REGION Network 13: Механізм крана
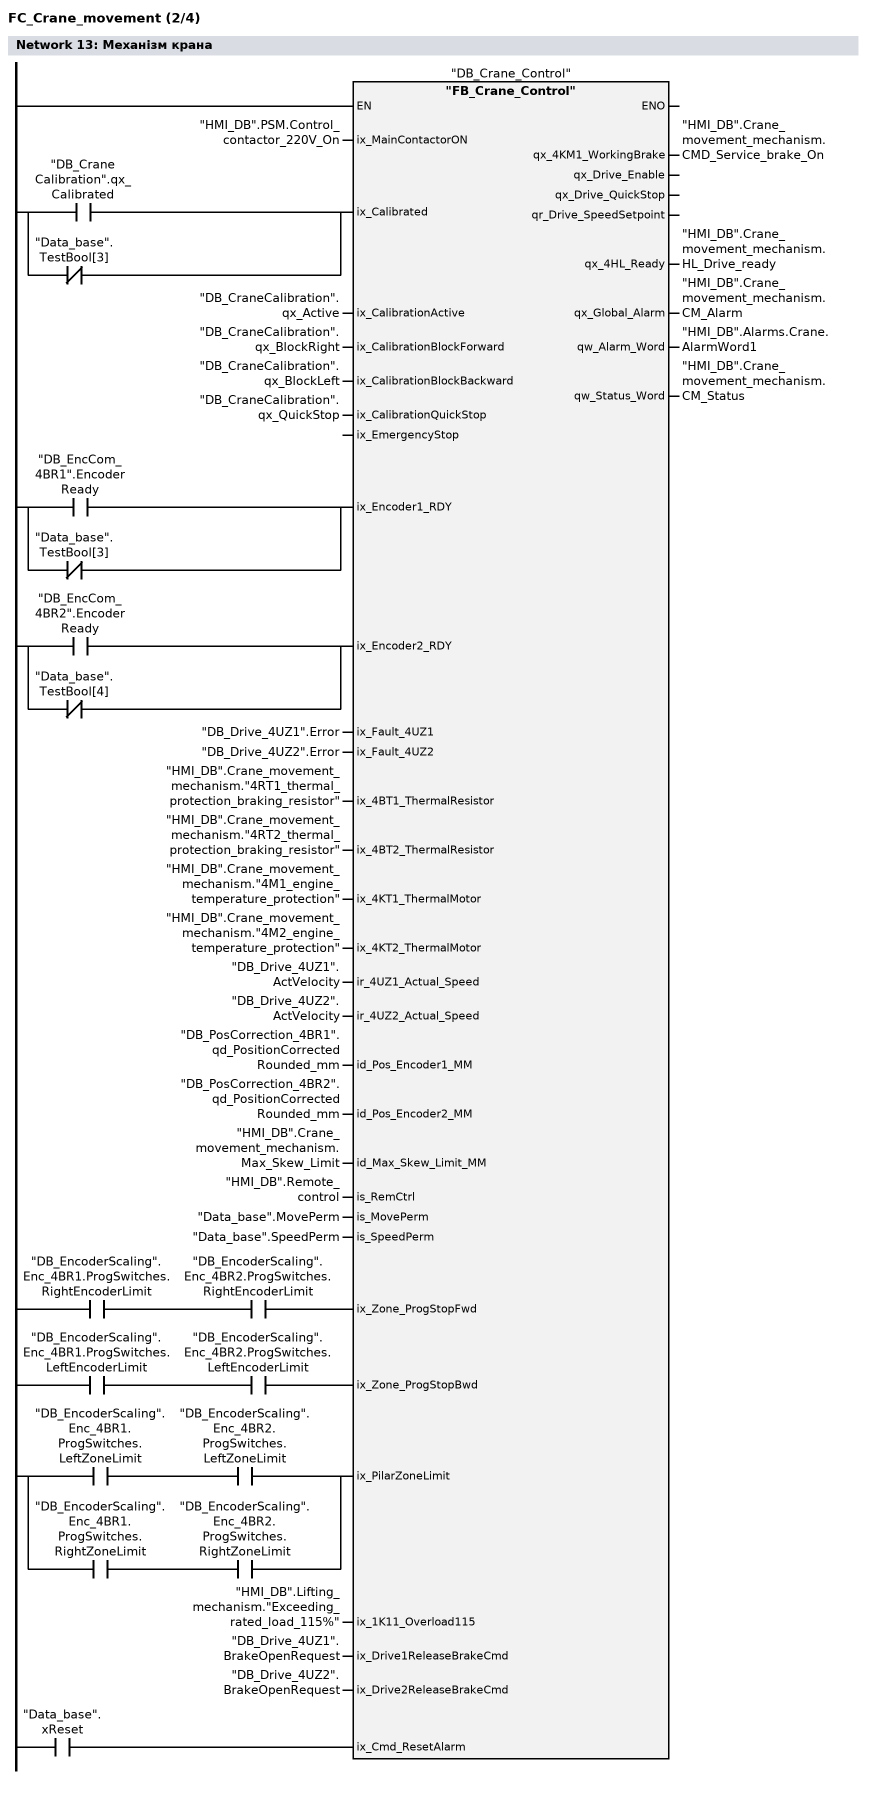
   RUNG wire#powerrail
      "DB_Crane_Control"(ix_Calibrated := wire#w1, ix_Encoder1_RDY := wire#w2, ix_Encoder2_RDY := wire#w3, ix_Zone_ProgStopFwd := wire#w4, ix_Zone_ProgStopBwd := wire#w5, ix_PilarZoneLimit := wire#w6, ix_Cmd_ResetAlarm := wire#w7, ix_MainContactorON := "HMI_DB".PSM.Control_contactor_220V_On, ix_CalibrationActive := "DB_CraneCalibration".qx_Active, ix_CalibrationBlockForward := "DB_CraneCalibration".qx_BlockRight, ix_CalibrationBlockBackward := "DB_CraneCalibration".qx_BlockLeft, ix_CalibrationQuickStop := "DB_CraneCalibration".qx_QuickStop, ix_EmergencyStop :=, ix_Fault_4UZ1 := "DB_Drive_4UZ1".Error, ix_Fault_4UZ2 := "DB_Drive_4UZ2".Error, ix_4BT1_ThermalResistor := "HMI_DB".Crane_movement_mechanism."4RT1_thermal_protection_braking_resistor", ix_4BT2_ThermalResistor := "HMI_DB".Crane_movement_mechanism."4RT2_thermal_protection_braking_resistor", ix_4KT1_ThermalMotor := "HMI_DB".Crane_movement_mechanism."4M1_engine_temperature_protection", ix_4KT2_ThermalMotor := "HMI_DB".Crane_movement_mechanism."4M2_engine_temperature_protection", ir_4UZ1_Actual_Speed := "DB_Drive_4UZ1".ActVelocity, ir_4UZ2_Actual_Speed := "DB_Drive_4UZ2".ActVelocity, id_Pos_Encoder1_MM := "DB_PosCorrection_4BR1".qd_PositionCorrectedRounded_mm, id_Pos_Encoder2_MM := "DB_PosCorrection_4BR2".qd_PositionCorrectedRounded_mm, id_Max_Skew_Limit_MM := "HMI_DB".Crane_movement_mechanism.Max_Skew_Limit, is_RemCtrl := "HMI_DB".Remote_control, is_MovePerm := "Data_base".MovePerm, is_SpeedPerm := "Data_base".SpeedPerm, ix_1K11_Overload115 := "HMI_DB".Lifting_mechanism."Exceeding_rated_load_115%", ix_Drive1ReleaseBrakeCmd := "DB_Drive_4UZ1".BrakeOpenRequest, ix_Drive2ReleaseBrakeCmd := "DB_Drive_4UZ2".BrakeOpenRequest, qx_4KM1_WorkingBrake => "HMI_DB".Crane_movement_mechanism.CMD_Service_brake_On, qx_Drive_Enable =>, qx_Drive_QuickStop =>, qr_Drive_SpeedSetpoint =>, qx_4HL_Ready => "HMI_DB".Crane_movement_mechanism.HL_Drive_ready, qx_Global_Alarm => "HMI_DB".Crane_movement_mechanism.CM_Alarm, qw_Alarm_Word => "HMI_DB".Alarms.Crane.AlarmWord1, qw_Status_Word => "HMI_DB".Crane_movement_mechanism.CM_Status)
   END_RUNG
   RUNG wire#powerrail
      Contact( "DB_CraneCalibration".qx_Calibrated )
   END_RUNG wire#w1
   RUNG wire#powerrail
      I_Contact( "Data_base".TestBool[3] )
   END_RUNG wire#w1
   RUNG wire#powerrail
      Contact( "DB_EncCom_4BR1".EncoderReady )
   END_RUNG wire#w2
   RUNG wire#powerrail
      I_Contact( "Data_base".TestBool[3] )
   END_RUNG wire#w2
   RUNG wire#powerrail
      Contact( "DB_EncCom_4BR2".EncoderReady )
   END_RUNG wire#w3
   RUNG wire#powerrail
      I_Contact( "Data_base".TestBool[4] )
   END_RUNG wire#w3
   RUNG wire#powerrail
      Contact( "DB_EncoderScaling".Enc_4BR1.ProgSwitches.RightEncoderLimit )
      Contact( "DB_EncoderScaling".Enc_4BR2.ProgSwitches.RightEncoderLimit )
   END_RUNG wire#w4
   RUNG wire#powerrail
      Contact( "DB_EncoderScaling".Enc_4BR1.ProgSwitches.LeftEncoderLimit )
      Contact( "DB_EncoderScaling".Enc_4BR2.ProgSwitches.LeftEncoderLimit )
   END_RUNG wire#w5
   RUNG wire#powerrail
      Contact( "DB_EncoderScaling".Enc_4BR1.ProgSwitches.LeftZoneLimit )
      Contact( "DB_EncoderScaling".Enc_4BR2.ProgSwitches.LeftZoneLimit )
   END_RUNG wire#w6
   RUNG wire#powerrail
      Contact( "DB_EncoderScaling".Enc_4BR1.ProgSwitches.RightZoneLimit )
      Contact( "DB_EncoderScaling".Enc_4BR2.ProgSwitches.RightZoneLimit )
   END_RUNG wire#w6
   RUNG wire#powerrail
      Contact( "Data_base".xReset )
   END_RUNG wire#w7
   // the same network as SCL:
   "DB_Crane_Control"(ix_MainContactorON := "HMI_DB".PSM.Control_contactor_220V_On,   // "FB_Crane_Control"
                      ix_Calibrated := "DB_CraneCalibration".qx_Calibrated OR NOT "Data_base".TestBool[3],
                      ix_CalibrationActive := "DB_CraneCalibration".qx_Active,
                      ix_CalibrationBlockForward := "DB_CraneCalibration".qx_BlockRight,
                      ix_CalibrationBlockBackward := "DB_CraneCalibration".qx_BlockLeft,
                      ix_CalibrationQuickStop := "DB_CraneCalibration".qx_QuickStop,
                      ix_Encoder1_RDY := "DB_EncCom_4BR1".EncoderReady OR NOT "Data_base".TestBool[3],
                      ix_Encoder2_RDY := "DB_EncCom_4BR2".EncoderReady OR NOT "Data_base".TestBool[4],
                      ix_Fault_4UZ1 := "DB_Drive_4UZ1".Error,
                      ix_Fault_4UZ2 := "DB_Drive_4UZ2".Error,
                      ix_4BT1_ThermalResistor := "HMI_DB".Crane_movement_mechanism."4RT1_thermal_protection_braking_resistor",
                      ix_4BT2_ThermalResistor := "HMI_DB".Crane_movement_mechanism."4RT2_thermal_protection_braking_resistor",
                      ix_4KT1_ThermalMotor := "HMI_DB".Crane_movement_mechanism."4M1_engine_temperature_protection",
                      ix_4KT2_ThermalMotor := "HMI_DB".Crane_movement_mechanism."4M2_engine_temperature_protection",
                      ir_4UZ1_Actual_Speed := "DB_Drive_4UZ1".ActVelocity,
                      ir_4UZ2_Actual_Speed := "DB_Drive_4UZ2".ActVelocity,
                      id_Pos_Encoder1_MM := "DB_PosCorrection_4BR1".qd_PositionCorrectedRounded_mm,
                      id_Pos_Encoder2_MM := "DB_PosCorrection_4BR2".qd_PositionCorrectedRounded_mm,
                      id_Max_Skew_Limit_MM := "HMI_DB".Crane_movement_mechanism.Max_Skew_Limit,
                      is_RemCtrl := "HMI_DB".Remote_control,
                      is_MovePerm := "Data_base".MovePerm,
                      is_SpeedPerm := "Data_base".SpeedPerm,
                      ix_Zone_ProgStopFwd := "DB_EncoderScaling".Enc_4BR1.ProgSwitches.RightEncoderLimit AND "DB_EncoderScaling".Enc_4BR2.ProgSwitches.RightEncoderLimit,
                      ix_Zone_ProgStopBwd := "DB_EncoderScaling".Enc_4BR1.ProgSwitches.LeftEncoderLimit AND "DB_EncoderScaling".Enc_4BR2.ProgSwitches.LeftEncoderLimit,
                      ix_PilarZoneLimit := ("DB_EncoderScaling".Enc_4BR1.ProgSwitches.LeftZoneLimit AND "DB_EncoderScaling".Enc_4BR2.ProgSwitches.LeftZoneLimit) OR ("DB_EncoderScaling".Enc_4BR1.ProgSwitches.RightZoneLimit AND "DB_EncoderScaling".Enc_4BR2.ProgSwitches.RightZoneLimit),
                      ix_1K11_Overload115 := "HMI_DB".Lifting_mechanism."Exceeding_rated_load_115%",
                      ix_Drive1ReleaseBrakeCmd := "DB_Drive_4UZ1".BrakeOpenRequest,
                      ix_Drive2ReleaseBrakeCmd := "DB_Drive_4UZ2".BrakeOpenRequest,
                      ix_Cmd_ResetAlarm := "Data_base".xReset,
                      qx_4KM1_WorkingBrake => "HMI_DB".Crane_movement_mechanism.CMD_Service_brake_On,
                      qx_4HL_Ready => "HMI_DB".Crane_movement_mechanism.HL_Drive_ready,
                      qx_Global_Alarm => "HMI_DB".Crane_movement_mechanism.CM_Alarm,
                      qw_Alarm_Word => "HMI_DB".Alarms.Crane.AlarmWord1,
                      qw_Status_Word => "HMI_DB".Crane_movement_mechanism.CM_Status);
END_REGION

REGION Network 14: Регістрація дій оператора
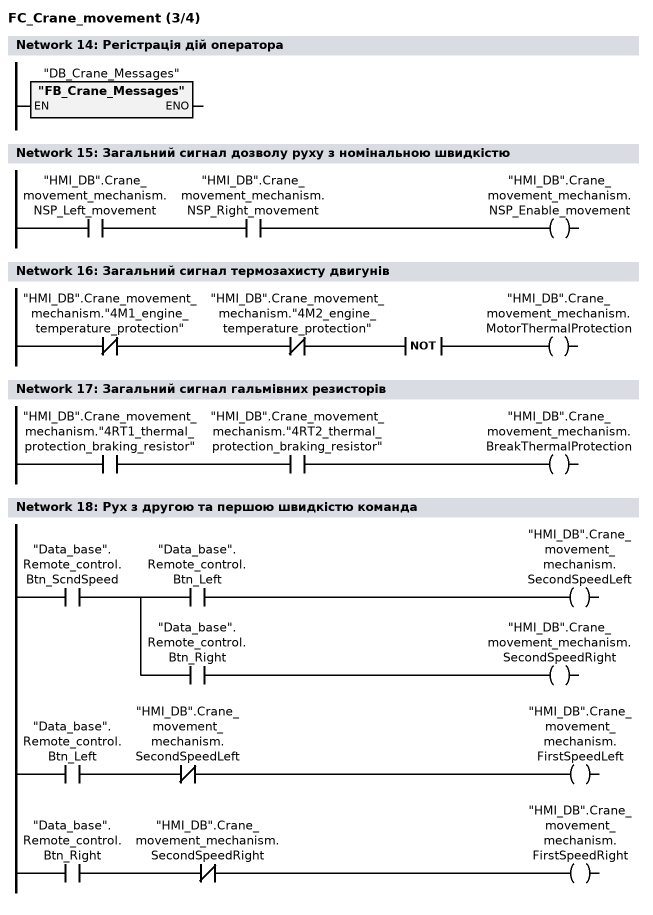
   RUNG wire#powerrail
      "DB_Crane_Messages"()
   END_RUNG
   // the same network as SCL:
   "DB_Crane_Messages"();   // "FB_Crane_Messages"
END_REGION

REGION Network 15: Загальний сигнал дозволу руху з номінальною швидкістю
   RUNG wire#powerrail
      Contact( "HMI_DB".Crane_movement_mechanism.NSP_Left_movement )
      Contact( "HMI_DB".Crane_movement_mechanism.NSP_Right_movement )
      Coil( "HMI_DB".Crane_movement_mechanism.NSP_Enable_movement )
   END_RUNG
   // the same network as SCL:
   "HMI_DB".Crane_movement_mechanism.NSP_Enable_movement := "HMI_DB".Crane_movement_mechanism.NSP_Left_movement AND "HMI_DB".Crane_movement_mechanism.NSP_Right_movement;
END_REGION

REGION Network 16: Загальний сигнал термозахисту двигунів
   RUNG wire#powerrail
      I_Contact( "HMI_DB".Crane_movement_mechanism."4M1_engine_temperature_protection" )
      I_Contact( "HMI_DB".Crane_movement_mechanism."4M2_engine_temperature_protection" )
      Not()
      Coil( "HMI_DB".Crane_movement_mechanism.MotorThermalProtection )
   END_RUNG
   // the same network as SCL:
   "HMI_DB".Crane_movement_mechanism.MotorThermalProtection := NOT (NOT "HMI_DB".Crane_movement_mechanism."4M1_engine_temperature_protection" AND NOT "HMI_DB".Crane_movement_mechanism."4M2_engine_temperature_protection");
END_REGION

REGION Network 17: Загальний сигнал гальмівних резисторів
   RUNG wire#powerrail
      Contact( "HMI_DB".Crane_movement_mechanism."4RT1_thermal_protection_braking_resistor" )
      Contact( "HMI_DB".Crane_movement_mechanism."4RT2_thermal_protection_braking_resistor" )
      Coil( "HMI_DB".Crane_movement_mechanism.BreakThermalProtection )
   END_RUNG
   // the same network as SCL:
   "HMI_DB".Crane_movement_mechanism.BreakThermalProtection := "HMI_DB".Crane_movement_mechanism."4RT1_thermal_protection_braking_resistor" AND "HMI_DB".Crane_movement_mechanism."4RT2_thermal_protection_braking_resistor";
END_REGION

REGION Network 18: Рух з другою та першою швидкістю команда
   RUNG wire#powerrail
      Contact( "Data_base".Remote_control.Btn_ScndSpeed )
      wire#w1
      Contact( "Data_base".Remote_control.Btn_Left )
      Coil( "HMI_DB".Crane_movement_mechanism.SecondSpeedLeft )
   END_RUNG
   RUNG wire#w1
      Contact( "Data_base".Remote_control.Btn_Right )
      Coil( "HMI_DB".Crane_movement_mechanism.SecondSpeedRight )
   END_RUNG
   RUNG wire#powerrail
      Contact( "Data_base".Remote_control.Btn_Left )
      I_Contact( "HMI_DB".Crane_movement_mechanism.SecondSpeedLeft )
      Coil( "HMI_DB".Crane_movement_mechanism.FirstSpeedLeft )
   END_RUNG
   RUNG wire#powerrail
      Contact( "Data_base".Remote_control.Btn_Right )
      I_Contact( "HMI_DB".Crane_movement_mechanism.SecondSpeedRight )
      Coil( "HMI_DB".Crane_movement_mechanism.FirstSpeedRight )
   END_RUNG
   // the same network as SCL:
   "HMI_DB".Crane_movement_mechanism.SecondSpeedLeft := "Data_base".Remote_control.Btn_ScndSpeed AND "Data_base".Remote_control.Btn_Left;
   "HMI_DB".Crane_movement_mechanism.SecondSpeedRight := "Data_base".Remote_control.Btn_ScndSpeed AND "Data_base".Remote_control.Btn_Right;
   "HMI_DB".Crane_movement_mechanism.FirstSpeedLeft := "Data_base".Remote_control.Btn_Left AND NOT "HMI_DB".Crane_movement_mechanism.SecondSpeedLeft;
   "HMI_DB".Crane_movement_mechanism.FirstSpeedRight := "Data_base".Remote_control.Btn_Right AND NOT "HMI_DB".Crane_movement_mechanism.SecondSpeedRight;
END_REGION

REGION Network 19: Формування попереджень калібровки
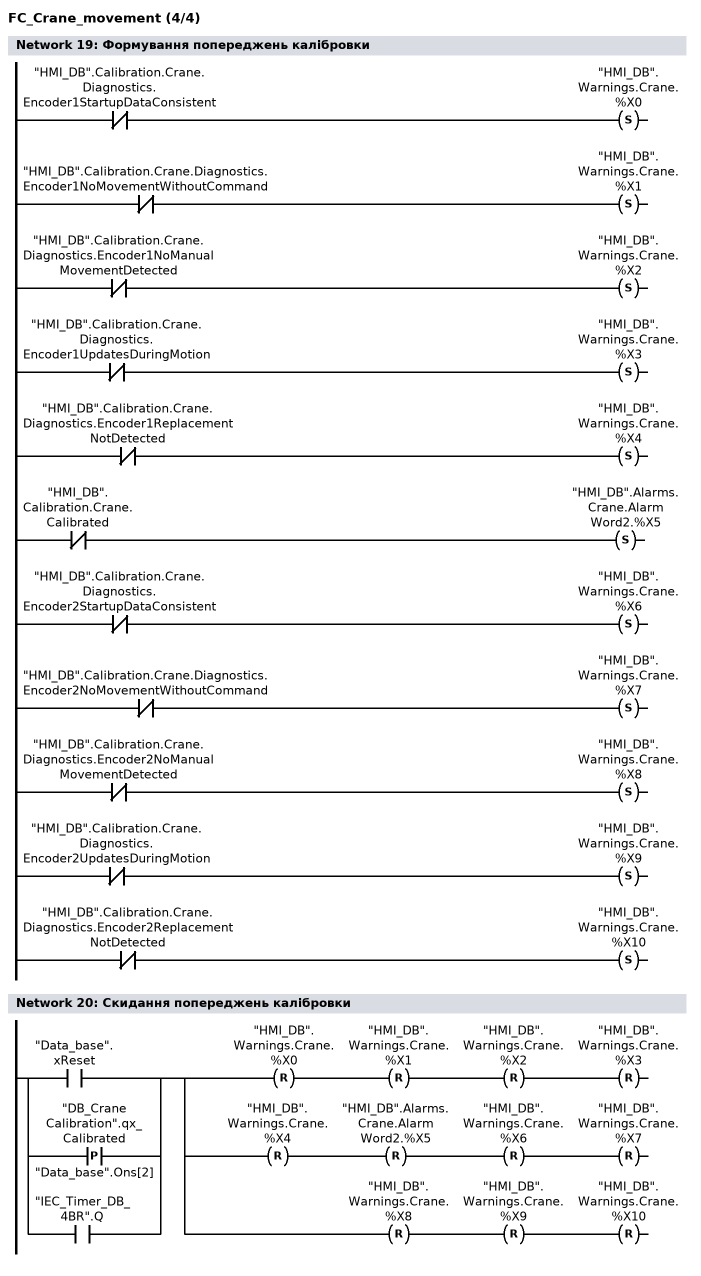
   RUNG wire#powerrail
      I_Contact( "HMI_DB".Calibration.Crane.Diagnostics.Encoder1StartupDataConsistent )
      S_Coil( "HMI_DB".Warnings.Crane.%X0 )
   END_RUNG
   RUNG wire#powerrail
      I_Contact( "HMI_DB".Calibration.Crane.Diagnostics.Encoder1NoMovementWithoutCommand )
      S_Coil( "HMI_DB".Warnings.Crane.%X1 )
   END_RUNG
   RUNG wire#powerrail
      I_Contact( "HMI_DB".Calibration.Crane.Diagnostics.Encoder1NoManualMovementDetected )
      S_Coil( "HMI_DB".Warnings.Crane.%X2 )
   END_RUNG
   RUNG wire#powerrail
      I_Contact( "HMI_DB".Calibration.Crane.Diagnostics.Encoder1UpdatesDuringMotion )
      S_Coil( "HMI_DB".Warnings.Crane.%X3 )
   END_RUNG
   RUNG wire#powerrail
      I_Contact( "HMI_DB".Calibration.Crane.Diagnostics.Encoder1ReplacementNotDetected )
      S_Coil( "HMI_DB".Warnings.Crane.%X4 )
   END_RUNG
   RUNG wire#powerrail
      I_Contact( "HMI_DB".Calibration.Crane.Calibrated )
      S_Coil( "HMI_DB".Alarms.Crane.AlarmWord2.%X5 )
   END_RUNG
   RUNG wire#powerrail
      I_Contact( "HMI_DB".Calibration.Crane.Diagnostics.Encoder2StartupDataConsistent )
      S_Coil( "HMI_DB".Warnings.Crane.%X6 )
   END_RUNG
   RUNG wire#powerrail
      I_Contact( "HMI_DB".Calibration.Crane.Diagnostics.Encoder2NoMovementWithoutCommand )
      S_Coil( "HMI_DB".Warnings.Crane.%X7 )
   END_RUNG
   RUNG wire#powerrail
      I_Contact( "HMI_DB".Calibration.Crane.Diagnostics.Encoder2NoManualMovementDetected )
      S_Coil( "HMI_DB".Warnings.Crane.%X8 )
   END_RUNG
   RUNG wire#powerrail
      I_Contact( "HMI_DB".Calibration.Crane.Diagnostics.Encoder2UpdatesDuringMotion )
      S_Coil( "HMI_DB".Warnings.Crane.%X9 )
   END_RUNG
   RUNG wire#powerrail
      I_Contact( "HMI_DB".Calibration.Crane.Diagnostics.Encoder2ReplacementNotDetected )
      S_Coil( "HMI_DB".Warnings.Crane.%X10 )
   END_RUNG
   // the same network as SCL:
   IF NOT "HMI_DB".Calibration.Crane.Diagnostics.Encoder1StartupDataConsistent THEN
       "HMI_DB".Warnings.Crane.%X0 := TRUE;
   END_IF;
   IF NOT "HMI_DB".Calibration.Crane.Diagnostics.Encoder1NoMovementWithoutCommand THEN
       "HMI_DB".Warnings.Crane.%X1 := TRUE;
   END_IF;
   IF NOT "HMI_DB".Calibration.Crane.Diagnostics.Encoder1NoManualMovementDetected THEN
       "HMI_DB".Warnings.Crane.%X2 := TRUE;
   END_IF;
   IF NOT "HMI_DB".Calibration.Crane.Diagnostics.Encoder1UpdatesDuringMotion THEN
       "HMI_DB".Warnings.Crane.%X3 := TRUE;
   END_IF;
   IF NOT "HMI_DB".Calibration.Crane.Diagnostics.Encoder1ReplacementNotDetected THEN
       "HMI_DB".Warnings.Crane.%X4 := TRUE;
   END_IF;
   IF NOT "HMI_DB".Calibration.Crane.Calibrated THEN "HMI_DB".Alarms.Crane.AlarmWord2.%X5 := TRUE; END_IF;
   IF NOT "HMI_DB".Calibration.Crane.Diagnostics.Encoder2StartupDataConsistent THEN
       "HMI_DB".Warnings.Crane.%X6 := TRUE;
   END_IF;
   IF NOT "HMI_DB".Calibration.Crane.Diagnostics.Encoder2NoMovementWithoutCommand THEN
       "HMI_DB".Warnings.Crane.%X7 := TRUE;
   END_IF;
   IF NOT "HMI_DB".Calibration.Crane.Diagnostics.Encoder2NoManualMovementDetected THEN
       "HMI_DB".Warnings.Crane.%X8 := TRUE;
   END_IF;
   IF NOT "HMI_DB".Calibration.Crane.Diagnostics.Encoder2UpdatesDuringMotion THEN
       "HMI_DB".Warnings.Crane.%X9 := TRUE;
   END_IF;
   IF NOT "HMI_DB".Calibration.Crane.Diagnostics.Encoder2ReplacementNotDetected THEN
       "HMI_DB".Warnings.Crane.%X10 := TRUE;
   END_IF;
END_REGION

REGION Network 20: Скидання попереджень калібровки
   RUNG wire#powerrail
      Contact( "Data_base".xReset )
      wire#w1
      R_Coil( "HMI_DB".Warnings.Crane.%X0 )
      R_Coil( "HMI_DB".Warnings.Crane.%X1 )
      R_Coil( "HMI_DB".Warnings.Crane.%X2 )
      R_Coil( "HMI_DB".Warnings.Crane.%X3 )
   END_RUNG
   RUNG wire#powerrail
      P_Contact(operand := "DB_CraneCalibration".qx_Calibrated, bit := "Data_base".Ons[2])
   END_RUNG wire#w1
   RUNG wire#powerrail
      Contact( "IEC_Timer_DB_4BR".Q )
   END_RUNG wire#w1
   RUNG wire#w1
      R_Coil( "HMI_DB".Warnings.Crane.%X4 )
      R_Coil( "HMI_DB".Alarms.Crane.AlarmWord2.%X5 )
      R_Coil( "HMI_DB".Warnings.Crane.%X6 )
      R_Coil( "HMI_DB".Warnings.Crane.%X7 )
   END_RUNG
   RUNG wire#w1
      R_Coil( "HMI_DB".Warnings.Crane.%X8 )
      R_Coil( "HMI_DB".Warnings.Crane.%X9 )
      R_Coil( "HMI_DB".Warnings.Crane.%X10 )
   END_RUNG
   // the same network as SCL:
   #_w1 := "DB_CraneCalibration".qx_Calibrated AND NOT "Data_base".Ons[2];   // rising edge of "DB_CraneCalibration".qx_Calibrated
   "Data_base".Ons[2] := "DB_CraneCalibration".qx_Calibrated;
   IF "Data_base".xReset OR #_w1 OR "IEC_Timer_DB_4BR".Q THEN
       "HMI_DB".Warnings.Crane.%X0 := FALSE;
       "HMI_DB".Warnings.Crane.%X1 := FALSE;
       "HMI_DB".Warnings.Crane.%X2 := FALSE;
       "HMI_DB".Warnings.Crane.%X3 := FALSE;
       "HMI_DB".Warnings.Crane.%X4 := FALSE;
       "HMI_DB".Alarms.Crane.AlarmWord2.%X5 := FALSE;
       "HMI_DB".Warnings.Crane.%X6 := FALSE;
       "HMI_DB".Warnings.Crane.%X7 := FALSE;
       "HMI_DB".Warnings.Crane.%X8 := FALSE;
       "HMI_DB".Warnings.Crane.%X9 := FALSE;
       "HMI_DB".Warnings.Crane.%X10 := FALSE;
   END_IF;
END_REGION
END_FUNCTION

// folder: 50_Drives

FUNCTION_BLOCK "FB_S120_Tel220"   // FB51, SCL
{ S7_Optimized_Access := 'TRUE' }
VERSION : 0.1
   VAR_INPUT
      EnableAxis : Bool := FALSE;   // Дозвіл роботи осі / ПЧ
      AckError : Bool := FALSE;   // Квітування аварії ПЧ, обробляється по фронту
      SimMode : Bool := FALSE;   // TRUE = режим симуляції, обмін з реальним ПЧ не виконується
      HWID_Tel220 : Hw_Io := 0;   // Hardware ID Telegram 220 для читання та запису PZD
      SpeedSp : Real := 0.0;   // Завдання швидкості, об/хв
      TorqueLimit : Real := 100.0;   // Обмеження моменту, %
      QuickStop : Bool := FALSE;   // Команда Quick Stop / OFF3
      CoastStop : Bool := FALSE;   // Команда Coast Stop / OFF2
      BrakesReleased : Bool := FALSE;   // Зворотний зв'язок: робоче та вбудоване гальма розгальмовані
      SimTelIn : "UDT_S120_Tel220_In";   // Симульована telegram від ПЧ
   END_VAR
   VAR_OUTPUT
      AxisEnabled : Bool := FALSE;   // ПЧ увімкнений та робота дозволена
      Lockout : Bool := FALSE;   // ПЧ не готовий до роботи або є заборона вмикання
      ActVelocity : Real := 0.0;   // Фактична швидкість, об/хв
      SpeedSetpointFb : Real := 0.0;   // Зворотний зв'язок по завданню швидкості, об/хв
      ActCurrent : Real := 0.0;   // Фактичний струм, А
      ActTorque : Real := 0.0;   // Фактичний момент, Н·м
      ActPower : Real := 0.0;   // Поточна активна потужність, кВт
      LoadPower : Real := 0.0;   // Завантаження механізму по потужності, %
      BrakeOpenRequest : Bool := FALSE;   // ПЧ запитує відкриття гальма
      Error : Bool := FALSE;   // Помилка драйвера або аварія ПЧ
      Status : Word := W#16#0000;   // Статус драйвера, бітове слово
      DiagId : Word := W#16#0000;   // Код діагностики драйвера / обміну
      FaultCode : Word := W#16#0000;   // Код аварії ПЧ
      WarningCode : Word := W#16#0000;   // Код попередження ПЧ
      TelOut : "UDT_S120_Tel220_Out";   // Сформована telegram PLC -> ПЧ, також для симулятора
   END_VAR
   VAR
      TelIn : "UDT_S120_Tel220_In";   // Остання прийнята telegram ПЧ -> PLC
      BrakeStatus : "UDT_S120_BrakeStatus";   // Розшифрований статус гальма з r1229
      ReadOk : Bool := FALSE;   // Читання telegram виконано без помилки
      WriteOk : Bool := FALSE;   // Запис telegram виконано без помилки
      ReadStatus : Int := 0;   // Код повернення DPRD_DAT
      WriteStatus : Int := 0;   // Код повернення DPWR_DAT
      ReadyToSwitchOn : Bool := FALSE;   // ПЧ готовий до вмикання
      ReadyToOperate : Bool := FALSE;   // ПЧ готовий до роботи
      OperationEnabled : Bool := FALSE;   // Робота ПЧ дозволена
      DriveFault : Bool := FALSE;   // Є аварія ПЧ
      DriveWarning : Bool := FALSE;   // Є попередження ПЧ
      NoCoastStopActive : Bool := FALSE;   // OFF2 не активний
      NoQuickStopActive : Bool := FALSE;   // OFF3 / Quick Stop не активний
      SwitchingOnInhibit : Bool := FALSE;   // Активна заборона вмикання
      ControlRequested : Bool := FALSE;   // ПЧ запитує керування від PLC
      RefSpeed_Rpm : Real := 1000.0;   // Опорна швидкість p2000, об/хв
      RefCurrent_A : Real := 1.0;   // Опорний струм p2002, А
      RefTorque_Nm : Real := 100.0;   // Опорний момент p2003, Н·м
      RefPower_kW : Real := 1.0;   // Опорна потужність p2004, кВт
      MotorRatedPower_kW : Real := 1.0;   // Номінальна потужність двигуна, кВт
      ResetFaultOld : Bool := FALSE;   // Попередній стан команди квітування аварії
      AckPulseCounter : Int := 0;   // Лічильник тривалості імпульсу квітування
      AckPulseCycles : Int := 10;   // Тривалість імпульсу квітування в циклах OB
   END_VAR
   VAR_TEMP
      ResetFaultPulse : Bool;   // Імпульс квітування аварії
      SpeedRawReal : Real;   // Завдання швидкості у сирому форматі telegram
      TorqueLimitRawReal : Real;   // Обмеження моменту у сирому форматі telegram
      TorqueLimitUsedPct : Real;   // Використане значення обмеження моменту
      AbsPower_kW : Real;   // Модуль активної потужності
   END_VAR
BEGIN
   // ============================================================
   // 1. Формування імпульсу квітування аварії
   // ============================================================

   IF #AckError AND NOT #ResetFaultOld THEN
       #AckPulseCounter := #AckPulseCycles;
   END_IF;

   #ResetFaultOld := #AckError;

   IF #AckPulseCounter > 0 THEN
       #ResetFaultPulse := TRUE;
       #AckPulseCounter := #AckPulseCounter - 1;
   ELSE
       #ResetFaultPulse := FALSE;
   END_IF;

   // ============================================================
   // 2. Формування вихідної telegram PLC -> ПЧ
   // ============================================================

   #TelOut.STW1_BM := W#16#0000;
   #TelOut.NSOLL_B := 0;
   #TelOut.STW2_BM := W#16#0000;
   #TelOut.M_ADD := 0;
   #TelOut.M_LIM := 0;
   #TelOut.USER_1 := W#16#0000;
   #TelOut.USER_2 := W#16#0000;
   #TelOut.USER_3 := W#16#0000;
   #TelOut.USER_4 := W#16#0000;

   // ============================================================
   // Feedback стану гальм для SINAMICS
   // Використовується механізмом підйому 1UZ1
   // ============================================================

   // PZD7, USER_1 bit 0:
   // робоче гальмо 1MB1 розгальмоване
   #TelOut.STW2_BM.%X12 := #BrakesReleased;
   #TelOut.STW2_BM.%X13 := NOT #BrakesReleased;
   // ============================================================

   // STW1_BM, базове керування PROFIdrive
   // Біт 01 = OFF2 не активний
   #TelOut.STW1_BM.%X1 := NOT #CoastStop;

   // Біт 02 = OFF3 / Quick Stop не активний
   #TelOut.STW1_BM.%X2 := NOT #QuickStop;

   // Біт 10 = керування від PLC
   #TelOut.STW1_BM.%X10 := TRUE;


       // Біт 09 = Enable Speed Controller
       #TelOut.STW2_BM.%X9 := TRUE;

   //IF #EnableAxis AND NOT #QuickStop AND NOT #CoastStop THEN
       // Біт 00 = ON / OFF1
       #TelOut.STW1_BM.%X0 :=#EnableAxis;

       // Біт 03 = дозвіл роботи
       #TelOut.STW1_BM.%X3 := TRUE;

       // Біт 04 = дозвіл генератора рампи
       #TelOut.STW1_BM.%X4 := TRUE;

       // Біт 05 = продовження роботи генератора рампи
       #TelOut.STW1_BM.%X5 := TRUE;


       // Біт 06 = дозвіл завдання швидкості
       #TelOut.STW1_BM.%X6 := TRUE;
   //END_IF;

   // Біт 07 = квітування аварії ПЧ, імпульсом
   #TelOut.STW1_BM.%X7 := #ResetFaultPulse;


   // ============================================================
   // 3. Масштабування завдання швидкості
   // NSOLL_B є 32-бітовим нормалізованим значенням.
   // 16#40000000 = 1073741824 = 100 % RefSpeed_Rpm
   // ============================================================

   IF #EnableAxis
       AND NOT #QuickStop
       AND NOT #CoastStop
       AND (#RefSpeed_Rpm > 0.0)
   THEN
       #SpeedRawReal := (#SpeedSp / #RefSpeed_Rpm) * 1073741824.0;

       IF #SpeedRawReal > 2147483647.0 THEN
           #SpeedRawReal := 2147483647.0;
       ELSIF #SpeedRawReal < -2147483648.0 THEN
           #SpeedRawReal := -2147483648.0;
       END_IF;

       #TelOut.NSOLL_B := REAL_TO_DINT(#SpeedRawReal);
   ELSE
       #TelOut.NSOLL_B := 0;
   END_IF;

   // ============================================================
   // 4. Обмеження моменту
   // ============================================================

   IF #TorqueLimit > 0.0 THEN
       #TorqueLimitUsedPct := #TorqueLimit;
   ELSE
       #TorqueLimitUsedPct := 100.0;
   END_IF;

   #TorqueLimitRawReal := (#TorqueLimitUsedPct / 100.0) * 16384.0;

   IF #TorqueLimitRawReal > 32767.0 THEN
       #TorqueLimitRawReal := 32767.0;
   ELSIF #TorqueLimitRawReal < 0.0 THEN
       #TorqueLimitRawReal := 0.0;
   END_IF;

   #TelOut.M_LIM := REAL_TO_INT(#TorqueLimitRawReal);


   // ============================================================
   // 5. Запис telegram PLC -> ПЧ
   // Один HWID_Tel220 використовується для запису та читання
   // ============================================================

   //IF #SimMode THEN
   //    #WriteStatus := 0;
   //    #WriteOk := TRUE;
   //ELSE
    //   #WriteStatus := DPWR_DAT(
    //                            LADDR := #HWID_Tel220,
   //                             RECORD := #TelOut
    //   );
    //   #WriteOk := (#WriteStatus = 0);
   //END_IF;

   #WriteStatus := DPWR_DAT(
                            LADDR := #HWID_Tel220,
                            RECORD := #TelOut
   );
   #WriteOk := (#WriteStatus = 0);

   // ============================================================
   // 6. Читання telegram ПЧ -> PLC або симуляція
   // Один HWID_Tel220 використовується для запису та читання
   // ============================================================

   //IF #SimMode THEN
    //   #TelIn := #SimTelIn;
    //   #ReadStatus := 0;
   //    #ReadOk := TRUE;
   //ELSE
    //   #ReadStatus := DPRD_DAT(
    //                           LADDR := #HWID_Tel220,
    //                           RECORD => #TelIn
    //   );

    //   #ReadOk := (#ReadStatus = 0);
   //END_IF;
   #ReadStatus := DPRD_DAT(
                           LADDR := #HWID_Tel220,
                           RECORD => #TelIn
   );

   #ReadOk := (#ReadStatus = 0);

   // ============================================================
   // 7. Декодування ZSW1_BM
   // ============================================================

   #ReadyToSwitchOn := #TelIn.ZSW1_BM.%X0;
   #ReadyToOperate := #TelIn.ZSW1_BM.%X1;
   #OperationEnabled := #TelIn.ZSW1_BM.%X2;
   #DriveFault := #TelIn.ZSW1_BM.%X3;
   #NoCoastStopActive := #TelIn.ZSW1_BM.%X4;
   #NoQuickStopActive := #TelIn.ZSW1_BM.%X5;
   #SwitchingOnInhibit := #TelIn.ZSW1_BM.%X6;
   #DriveWarning := #TelIn.ZSW1_BM.%X7;
   #ControlRequested := #TelIn.ZSW1_BM.%X9;


   // ============================================================
   // 8. Основні статуси для зовнішньої логіки
   // ============================================================

   #AxisEnabled := #ReadOk
   AND #WriteOk
   AND #OperationEnabled
   AND NOT #DriveFault;

   #Lockout := (NOT #ReadOk)
   OR (NOT #WriteOk)
   OR #DriveFault
   OR #SwitchingOnInhibit
   OR (NOT #NoCoastStopActive)
   OR (NOT #NoQuickStopActive);

   #Error := (NOT #ReadOk)
   OR (NOT #WriteOk)
   OR #DriveFault;


   // ============================================================
   // 9. Коди fault / warning
   // ============================================================

   #FaultCode := #TelIn.FAULT_CODE;
   #WarningCode := #TelIn.WARN_CODE;


   // ============================================================
   // 10. Масштабування фактичних значень
   // ============================================================

   #ActVelocity := 0.0;
   #SpeedSetpointFb := 0.0;
   #ActCurrent := 0.0;
   #ActTorque := 0.0;
   #ActPower := 0.0;
   #LoadPower := 0.0;
   #AbsPower_kW := 0.0;

   IF #RefSpeed_Rpm > 0.0 THEN
       #ActVelocity := (INT_TO_REAL(#TelIn.NIST_A) / 16384.0) * #RefSpeed_Rpm;
       #SpeedSetpointFb := (INT_TO_REAL(#TelIn.NSET_FB) / 16384.0) * #RefSpeed_Rpm;
   END_IF;

   IF #RefCurrent_A > 0.0 THEN
       #ActCurrent := (INT_TO_REAL(#TelIn.IAIST) / 16384.0) * #RefCurrent_A;
   END_IF;

   IF #RefTorque_Nm > 0.0 THEN
       #ActTorque := (INT_TO_REAL(#TelIn.MIST) / 16384.0) * #RefTorque_Nm;
   END_IF;

   IF #RefPower_kW > 0.0 THEN
       #ActPower := (INT_TO_REAL(#TelIn.P_ACT) / 16384.0) * #RefPower_kW;
   END_IF;

   IF #ActPower < 0.0 THEN
       #AbsPower_kW := - #ActPower;
   ELSE
       #AbsPower_kW := #ActPower;
   END_IF;

   IF #MotorRatedPower_kW > 0.0 THEN
       #LoadPower := (#AbsPower_kW / #MotorRatedPower_kW) * 100.0;
   END_IF;

   // ============================================================
   // 11. Декодування статусу гальма з BRAKE_STATUS / r1229
   // ============================================================

   #BrakeStatus.CommandOpenBrake := #TelIn.BRAKE_STATUS.%X1;
   #BrakeStatus.PulseEnableExtendedBrakeControl := #TelIn.BRAKE_STATUS.%X3;
   #BrakeStatus.BrakeDoesNotOpen := #TelIn.BRAKE_STATUS.%X4;
   #BrakeStatus.BrakeDoesNotClose := #TelIn.BRAKE_STATUS.%X5;
   #BrakeStatus.BrakeThresholdExceeded := #TelIn.BRAKE_STATUS.%X6;
   #BrakeStatus.BrakeThresholdUndershot := #TelIn.BRAKE_STATUS.%X7;
   #BrakeStatus.BrakeMonitoringTimeExpired := #TelIn.BRAKE_STATUS.%X8;
   #BrakeStatus.PulseEnableRequestMissing := #TelIn.BRAKE_STATUS.%X9;
   #BrakeStatus.BrakeOrLogicResult := #TelIn.BRAKE_STATUS.%X10;
   #BrakeStatus.BrakeAndLogicResult := #TelIn.BRAKE_STATUS.%X11;

   #BrakeOpenRequest := #BrakeStatus.CommandOpenBrake;


   // ============================================================
   // 12. Формування Status
   // ============================================================

   #Status := W#16#0000;

   #Status.%X0 := #ReadOk;                  // Біт 0: читання telegram OK
   #Status.%X1 := #WriteOk;                 // Біт 1: запис telegram OK
   #Status.%X2 := #AxisEnabled;             // Біт 2: ПЧ у роботі
   #Status.%X3 := #Lockout;                 // Біт 3: блокування / неготовність
   #Status.%X4 := #DriveFault;              // Біт 4: аварія ПЧ
   #Status.%X5 := #DriveWarning;            // Біт 5: попередження ПЧ
   #Status.%X6 := #BrakeOpenRequest;        // Біт 6: ПЧ запитує відкриття гальма
   #Status.%X7 := #SimMode;                 // Біт 7: активний режим симуляції
   #Status.%X8 := #SwitchingOnInhibit;      // Біт 8: заборона вмикання
   #Status.%X9 := #ControlRequested;        // Біт 9: ПЧ запитує керування від PLC


   // ============================================================
   // 13. Формування DiagId
   // ============================================================

   IF NOT #ReadOk THEN
       #DiagId := W#16#8201;                // Помилка читання telegram
   ELSIF NOT #WriteOk THEN
       #DiagId := W#16#8202;                // Помилка запису telegram
   ELSIF #DriveFault THEN
       #DiagId := W#16#8401;                // Аварія ПЧ
   ELSIF #SwitchingOnInhibit THEN
       #DiagId := W#16#8402;                // Активна заборона вмикання
   ELSIF NOT #EnableAxis THEN
       #DiagId := W#16#7000;                // Драйвер не увімкнений
   ELSE
       #DiagId := W#16#0000;                // Немає помилок
   END_IF;
END_FUNCTION_BLOCK

FUNCTION_BLOCK "FB_S120_Tel390_CU"   // FB52, SCL
{ S7_Optimized_Access := 'TRUE' }
VERSION : 0.1
   VAR_INPUT
      Enable : Bool := TRUE;   // Дозвіл роботи драйвера CU
      AckError : Bool := FALSE;   // Квітування помилки CU, обробляється по фронту
      SimMode : Bool := FALSE;   // TRUE = режим симуляції, обмін з реальною CU не виконується
      HWID_Tel390 : Hw_Io := 0;   // Hardware ID Telegram 390 для читання та запису PZD
      SimTelIn : "UDT_S120_Tel390_CU_In";   // Симульована telegram CU -> PLC
   END_VAR
   VAR_OUTPUT
      CommOk : Bool := FALSE;   // Обмін з CU справний або активний режим симуляції
      Fault : Bool := FALSE;   // CU повідомляє активну помилку
      Warning : Bool := FALSE;   // CU повідомляє активне попередження
      Error : Bool := FALSE;   // Помилка драйвера, комунікації або fault CU
      Status : Word := W#16#0000;   // Статус драйвера CU, бітове слово
      DiagId : Word := W#16#0000;   // Код діагностики драйвера CU
      CU_StatusWord : Word := W#16#0000;   // Сире статусне слово CU, PZD1
      CU_DiagCode : Word := W#16#0000;   // Діагностичне слово / код помилки або попередження CU, PZD2
      TelOut : "UDT_S120_Tel390_CU_Out";   // Сформована telegram PLC -> CU, також для симулятора
   END_VAR
   VAR
      TelIn : "UDT_S120_Tel390_CU_In";   // Остання прийнята telegram CU -> PLC
      StatusBits : "UDT_S120_Tel390_CU_ZSW1_Bits";   // Розшифровані біти статусного слова CU_ZSW1
      ReadOk : Bool := FALSE;   // Читання telegram виконано без помилки
      WriteOk : Bool := FALSE;   // Запис telegram виконано без помилки
      ReadStatus : Int := 0;   // Код повернення DPRD_DAT
      WriteStatus : Int := 0;   // Код повернення DPWR_DAT
      AckErrorOld : Bool := FALSE;   // Попередній стан команди квітування помилки
      AckPulseCounter : Int := 0;   // Лічильник тривалості імпульсу квітування
      AckPulseCycles : Int := 10;   // Тривалість імпульсу квітування в циклах OB
   END_VAR
   VAR_TEMP
      AckErrorPulse : Bool;   // Імпульс квітування помилки CU
   END_VAR
BEGIN
   // ============================================================
   // 1. Імпульс квітування помилки
   // ============================================================

   IF #AckError AND NOT #AckErrorOld THEN
       #AckPulseCounter := #AckPulseCycles;
   END_IF;

   #AckErrorOld := #AckError;

   IF #AckPulseCounter > 0 THEN
       #AckErrorPulse := TRUE;
       #AckPulseCounter := #AckPulseCounter - 1;
   ELSE
       #AckErrorPulse := FALSE;
   END_IF;


   // ============================================================
   // 2. Формування telegram PLC -> CU
   // Керування CU не використовується.
   // Використовуємо тільки:
   // - CU_STW1.%X10 = Master control by PLC / Remote control from PLC
   // - CU_STW1.%X7  = квітування помилки CU, імпульсом
   // ============================================================

   #TelOut.CU_STW1 := W#16#0000;
   #TelOut.CU_CTRL2 := W#16#0000;

   // Біт 10 = Remote control / Master control by PLC.
   // Тримати TRUE, коли драйвер CU увімкнений.
   #TelOut.CU_STW1.%X10 := #Enable;

   // Біт 7 = квітування помилки CU, імпульсом.
   #TelOut.CU_STW1.%X7 := #AckErrorPulse;


   // ============================================================
   // 3. Якщо драйвер вимкнений
   // ============================================================

   IF NOT #Enable THEN
       #ReadOk := FALSE;
       #WriteOk := FALSE;
       #CommOk := FALSE;

       #Fault := FALSE;
       #Warning := FALSE;
       #Error := FALSE;

       #CU_StatusWord := W#16#0000;
       #CU_DiagCode := W#16#0000;

       #Status := W#16#0000;
       #DiagId := W#16#7000;       // Драйвер CU вимкнений

       RETURN;
   END_IF;


   // ============================================================
   // 4. Запис telegram PLC -> CU
   // Один HWID_Tel390 використовується для запису та читання
   // ============================================================

   IF #SimMode THEN
       #WriteStatus := 0;
       #WriteOk := TRUE;
   ELSE
       #WriteStatus := DPWR_DAT(
                                LADDR := #HWID_Tel390,
                                RECORD := #TelOut
       );

       #WriteOk := (#WriteStatus = 0);
   END_IF;


   // ============================================================
   // 5. Читання telegram CU -> PLC або симуляція
   // Один HWID_Tel390 використовується для запису та читання
   // ============================================================

   IF #SimMode THEN
       #TelIn := #SimTelIn;
       #ReadStatus := 0;
       #ReadOk := TRUE;
   ELSE
       #ReadStatus := DPRD_DAT(
                               LADDR := #HWID_Tel390,
                               RECORD => #TelIn
       );

       #ReadOk := (#ReadStatus = 0);
   END_IF;


   // ============================================================
   // 6. Комунікація
   // ============================================================

   #CommOk := #ReadOk AND #WriteOk;


   // ============================================================
   // 7. Сирі слова telegram
   // ============================================================

   #CU_StatusWord := #TelIn.CU_ZSW1;
   #CU_DiagCode := #TelIn.CU_DIAG_CODE;


   // ============================================================
   // 8. Декодування CU_ZSW1
   // ============================================================

   #StatusBits.ReadyToSwitchOn := #TelIn.CU_ZSW1.%X0;
   #StatusBits.ReadyToOperate := #TelIn.CU_ZSW1.%X1;
   #StatusBits.OperationEnabled := #TelIn.CU_ZSW1.%X2;
   #StatusBits.FaultActive := #TelIn.CU_ZSW1.%X3;
   #StatusBits.NoCoastStopActive := #TelIn.CU_ZSW1.%X4;
   #StatusBits.NoQuickStopActive := #TelIn.CU_ZSW1.%X5;
   #StatusBits.SwitchingOnInhibit := #TelIn.CU_ZSW1.%X6;
   #StatusBits.WarningActive := #TelIn.CU_ZSW1.%X7;
   #StatusBits.Bit08 := #TelIn.CU_ZSW1.%X8;
   #StatusBits.ControlRequested := #TelIn.CU_ZSW1.%X9;
   #StatusBits.Bit10 := #TelIn.CU_ZSW1.%X10;
   #StatusBits.Bit11 := #TelIn.CU_ZSW1.%X11;
   #StatusBits.Bit12 := #TelIn.CU_ZSW1.%X12;
   #StatusBits.Bit13 := #TelIn.CU_ZSW1.%X13;
   #StatusBits.Bit14 := #TelIn.CU_ZSW1.%X14;
   #StatusBits.Bit15 := #TelIn.CU_ZSW1.%X15;


   // ============================================================
   // 9. Основні статуси CU
   // ============================================================

   #Fault := #StatusBits.FaultActive;
   #Warning := #StatusBits.WarningActive;

   #Error := (NOT #ReadOk)
   OR (NOT #WriteOk)
   OR #Fault;


   // ============================================================
   // 10. Формування Status
   // ============================================================

   #Status := W#16#0000;

   #Status.%X0 := #ReadOk;                         // Біт 0: читання telegram OK
   #Status.%X1 := #WriteOk;                        // Біт 1: запис telegram OK
   #Status.%X2 := #CommOk;                         // Біт 2: обмін з CU OK
   #Status.%X3 := #Fault;                          // Біт 3: fault CU
   #Status.%X4 := #Warning;                        // Біт 4: warning CU
   #Status.%X5 := #StatusBits.SwitchingOnInhibit;  // Біт 5: заборона / блокування CU
   #Status.%X6 := #StatusBits.ControlRequested;    // Біт 6: CU запитує керування від PLC
   #Status.%X7 := #SimMode;                        // Біт 7: активний режим симуляції


   // ============================================================
   // 11. Формування DiagId
   // ============================================================

   IF NOT #ReadOk THEN
       #DiagId := W#16#8201;          // Помилка читання telegram CU
   ELSIF NOT #WriteOk THEN
       #DiagId := W#16#8202;          // Помилка запису telegram CU
   ELSIF #Fault THEN
       #DiagId := W#16#8401;          // CU повідомляє fault
   ELSIF #Warning THEN
       #DiagId := W#16#8402;          // CU повідомляє warning
   ELSE
       #DiagId := W#16#0000;          // Немає помилок
   END_IF;
END_FUNCTION_BLOCK

FUNCTION "FC_Drives_Call" : Void   // FC50, LAD
TITLE = Комунікація з приводами
{ S7_Optimized_Access := 'TRUE' }
VERSION : 0.1
BEGIN

REGION Network 2: Ресет помилок
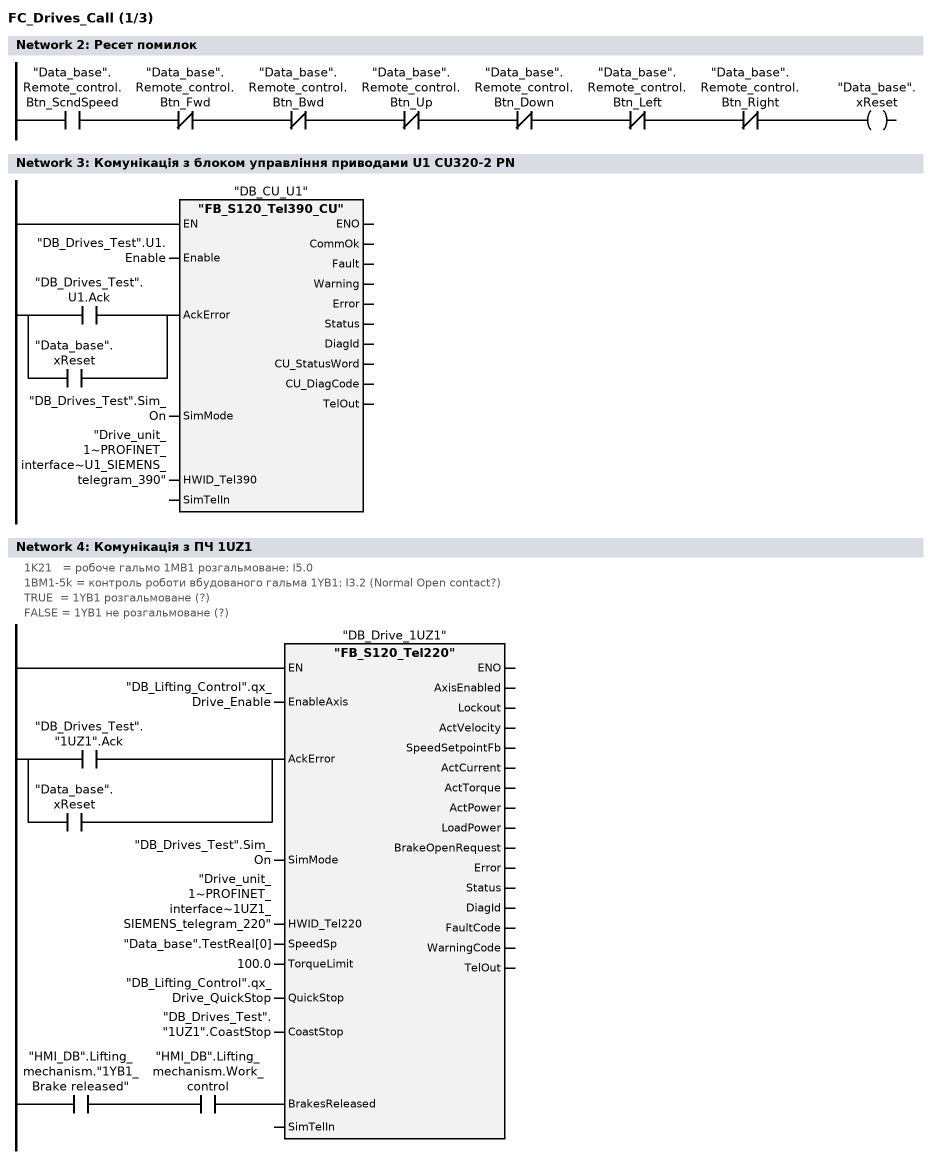
   RUNG wire#powerrail
      Contact( "Data_base".Remote_control.Btn_ScndSpeed )
      I_Contact( "Data_base".Remote_control.Btn_Fwd )
      I_Contact( "Data_base".Remote_control.Btn_Bwd )
      I_Contact( "Data_base".Remote_control.Btn_Up )
      I_Contact( "Data_base".Remote_control.Btn_Down )
      I_Contact( "Data_base".Remote_control.Btn_Left )
      I_Contact( "Data_base".Remote_control.Btn_Right )
      Coil( "Data_base".xReset )
   END_RUNG
   // the same network as SCL:
   "Data_base".xReset := "Data_base".Remote_control.Btn_ScndSpeed AND NOT "Data_base".Remote_control.Btn_Fwd AND NOT "Data_base".Remote_control.Btn_Bwd AND NOT "Data_base".Remote_control.Btn_Up AND NOT "Data_base".Remote_control.Btn_Down AND NOT "Data_base".Remote_control.Btn_Left AND NOT "Data_base".Remote_control.Btn_Right;
END_REGION

REGION Network 3: Комунікація з блоком управління приводами U1 CU320-2 PN
   RUNG wire#powerrail
      "DB_CU_U1"(AckError := wire#w1, Enable := "DB_Drives_Test".U1.Enable, SimMode := "DB_Drives_Test".Sim_On, HWID_Tel390 := "Drive_unit_1~PROFINET_interface~U1_SIEMENS_telegram_390", SimTelIn :=, CommOk =>, Fault =>, Warning =>, Error =>, Status =>, DiagId =>, CU_StatusWord =>, CU_DiagCode =>, TelOut =>)
   END_RUNG
   RUNG wire#powerrail
      Contact( "DB_Drives_Test".U1.Ack )
   END_RUNG wire#w1
   RUNG wire#powerrail
      Contact( "Data_base".xReset )
   END_RUNG wire#w1
   // the same network as SCL:
   "DB_CU_U1"(Enable := "DB_Drives_Test".U1.Enable,   // "FB_S120_Tel390_CU"
              AckError := "DB_Drives_Test".U1.Ack OR "Data_base".xReset,
              SimMode := "DB_Drives_Test".Sim_On,
              HWID_Tel390 := "Drive_unit_1~PROFINET_interface~U1_SIEMENS_telegram_390");
END_REGION

REGION Network 4: Комунікація з ПЧ 1UZ1
   // 1K21   = робоче гальмо 1MB1 розгальмоване: I5.0
   // 1BM1-5k = контроль роботи вбудованого гальма 1YB1: I3.2 (Normal Open contact?)
   // TRUE  = 1YB1 розгальмоване (?)
   // FALSE = 1YB1 не розгальмоване (?)
   RUNG wire#powerrail
      "DB_Drive_1UZ1"(AckError := wire#w1, BrakesReleased := wire#w2, EnableAxis := "DB_Lifting_Control".qx_Drive_Enable, SimMode := "DB_Drives_Test".Sim_On, HWID_Tel220 := "Drive_unit_1~PROFINET_interface~1UZ1_SIEMENS_telegram_220", SpeedSp := "Data_base".TestReal[0], TorqueLimit := 100.0, QuickStop := "DB_Lifting_Control".qx_Drive_QuickStop, CoastStop := "DB_Drives_Test"."1UZ1".CoastStop, SimTelIn :=, AxisEnabled =>, Lockout =>, ActVelocity =>, SpeedSetpointFb =>, ActCurrent =>, ActTorque =>, ActPower =>, LoadPower =>, BrakeOpenRequest =>, Error =>, Status =>, DiagId =>, FaultCode =>, WarningCode =>, TelOut =>)
   END_RUNG
   RUNG wire#powerrail
      Contact( "DB_Drives_Test"."1UZ1".Ack )
   END_RUNG wire#w1
   RUNG wire#powerrail
      Contact( "Data_base".xReset )
   END_RUNG wire#w1
   RUNG wire#powerrail
      Contact( "HMI_DB".Lifting_mechanism."1YB1_Brake released" )
      Contact( "HMI_DB".Lifting_mechanism.Work_control )
   END_RUNG wire#w2
   // the same network as SCL:
   "DB_Drive_1UZ1"(EnableAxis := "DB_Lifting_Control".qx_Drive_Enable,   // "FB_S120_Tel220"
                   AckError := "DB_Drives_Test"."1UZ1".Ack OR "Data_base".xReset,
                   SimMode := "DB_Drives_Test".Sim_On,
                   HWID_Tel220 := "Drive_unit_1~PROFINET_interface~1UZ1_SIEMENS_telegram_220",
                   SpeedSp := "Data_base".TestReal[0],
                   TorqueLimit := 100.0,
                   QuickStop := "DB_Lifting_Control".qx_Drive_QuickStop,
                   CoastStop := "DB_Drives_Test"."1UZ1".CoastStop,
                   BrakesReleased := "HMI_DB".Lifting_mechanism."1YB1_Brake released" AND "HMI_DB".Lifting_mechanism.Work_control);
END_REGION

REGION Network 5: Комунікація з ПЧ 3UZ1
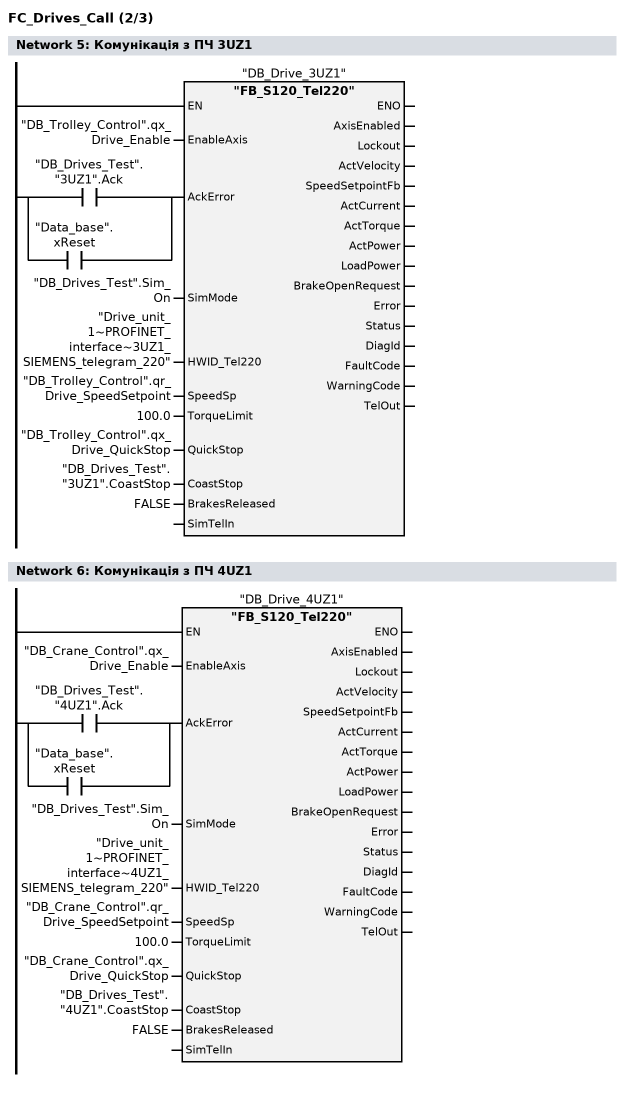
   RUNG wire#powerrail
      "DB_Drive_3UZ1"(AckError := wire#w1, EnableAxis := "DB_Trolley_Control".qx_Drive_Enable, SimMode := "DB_Drives_Test".Sim_On, HWID_Tel220 := "Drive_unit_1~PROFINET_interface~3UZ1_SIEMENS_telegram_220", SpeedSp := "DB_Trolley_Control".qr_Drive_SpeedSetpoint, TorqueLimit := 100.0, QuickStop := "DB_Trolley_Control".qx_Drive_QuickStop, CoastStop := "DB_Drives_Test"."3UZ1".CoastStop, BrakesReleased := FALSE, SimTelIn :=, AxisEnabled =>, Lockout =>, ActVelocity =>, SpeedSetpointFb =>, ActCurrent =>, ActTorque =>, ActPower =>, LoadPower =>, BrakeOpenRequest =>, Error =>, Status =>, DiagId =>, FaultCode =>, WarningCode =>, TelOut =>)
   END_RUNG
   RUNG wire#powerrail
      Contact( "DB_Drives_Test"."3UZ1".Ack )
   END_RUNG wire#w1
   RUNG wire#powerrail
      Contact( "Data_base".xReset )
   END_RUNG wire#w1
   // the same network as SCL:
   "DB_Drive_3UZ1"(EnableAxis := "DB_Trolley_Control".qx_Drive_Enable,   // "FB_S120_Tel220"
                   AckError := "DB_Drives_Test"."3UZ1".Ack OR "Data_base".xReset,
                   SimMode := "DB_Drives_Test".Sim_On,
                   HWID_Tel220 := "Drive_unit_1~PROFINET_interface~3UZ1_SIEMENS_telegram_220",
                   SpeedSp := "DB_Trolley_Control".qr_Drive_SpeedSetpoint,
                   TorqueLimit := 100.0,
                   QuickStop := "DB_Trolley_Control".qx_Drive_QuickStop,
                   CoastStop := "DB_Drives_Test"."3UZ1".CoastStop,
                   BrakesReleased := FALSE);
END_REGION

REGION Network 6: Комунікація з ПЧ 4UZ1
   RUNG wire#powerrail
      "DB_Drive_4UZ1"(AckError := wire#w1, EnableAxis := "DB_Crane_Control".qx_Drive_Enable, SimMode := "DB_Drives_Test".Sim_On, HWID_Tel220 := "Drive_unit_1~PROFINET_interface~4UZ1_SIEMENS_telegram_220", SpeedSp := "DB_Crane_Control".qr_Drive_SpeedSetpoint, TorqueLimit := 100.0, QuickStop := "DB_Crane_Control".qx_Drive_QuickStop, CoastStop := "DB_Drives_Test"."4UZ1".CoastStop, BrakesReleased := FALSE, SimTelIn :=, AxisEnabled =>, Lockout =>, ActVelocity =>, SpeedSetpointFb =>, ActCurrent =>, ActTorque =>, ActPower =>, LoadPower =>, BrakeOpenRequest =>, Error =>, Status =>, DiagId =>, FaultCode =>, WarningCode =>, TelOut =>)
   END_RUNG
   RUNG wire#powerrail
      Contact( "DB_Drives_Test"."4UZ1".Ack )
   END_RUNG wire#w1
   RUNG wire#powerrail
      Contact( "Data_base".xReset )
   END_RUNG wire#w1
   // the same network as SCL:
   "DB_Drive_4UZ1"(EnableAxis := "DB_Crane_Control".qx_Drive_Enable,   // "FB_S120_Tel220"
                   AckError := "DB_Drives_Test"."4UZ1".Ack OR "Data_base".xReset,
                   SimMode := "DB_Drives_Test".Sim_On,
                   HWID_Tel220 := "Drive_unit_1~PROFINET_interface~4UZ1_SIEMENS_telegram_220",
                   SpeedSp := "DB_Crane_Control".qr_Drive_SpeedSetpoint,
                   TorqueLimit := 100.0,
                   QuickStop := "DB_Crane_Control".qx_Drive_QuickStop,
                   CoastStop := "DB_Drives_Test"."4UZ1".CoastStop,
                   BrakesReleased := FALSE);
END_REGION

REGION Network 7: Комунікація з ПЧ 4UZ2
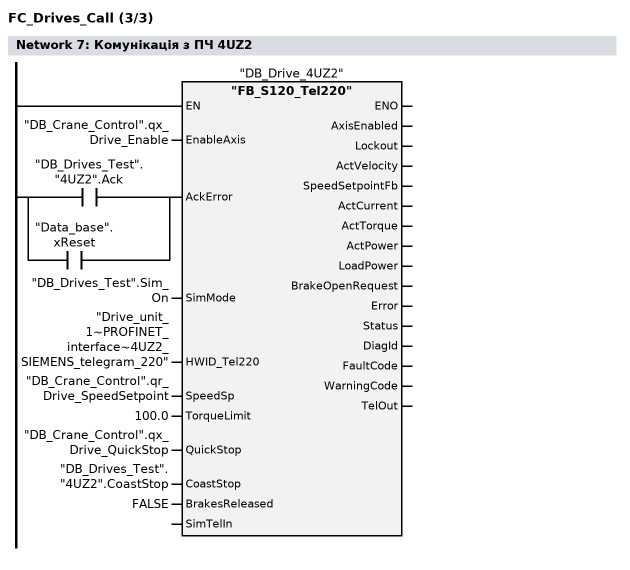
   RUNG wire#powerrail
      "DB_Drive_4UZ2"(AckError := wire#w1, EnableAxis := "DB_Crane_Control".qx_Drive_Enable, SimMode := "DB_Drives_Test".Sim_On, HWID_Tel220 := "Drive_unit_1~PROFINET_interface~4UZ2_SIEMENS_telegram_220", SpeedSp := "DB_Crane_Control".qr_Drive_SpeedSetpoint, TorqueLimit := 100.0, QuickStop := "DB_Crane_Control".qx_Drive_QuickStop, CoastStop := "DB_Drives_Test"."4UZ2".CoastStop, BrakesReleased := FALSE, SimTelIn :=, AxisEnabled =>, Lockout =>, ActVelocity =>, SpeedSetpointFb =>, ActCurrent =>, ActTorque =>, ActPower =>, LoadPower =>, BrakeOpenRequest =>, Error =>, Status =>, DiagId =>, FaultCode =>, WarningCode =>, TelOut =>)
   END_RUNG
   RUNG wire#powerrail
      Contact( "DB_Drives_Test"."4UZ2".Ack )
   END_RUNG wire#w1
   RUNG wire#powerrail
      Contact( "Data_base".xReset )
   END_RUNG wire#w1
   // the same network as SCL:
   "DB_Drive_4UZ2"(EnableAxis := "DB_Crane_Control".qx_Drive_Enable,   // "FB_S120_Tel220"
                   AckError := "DB_Drives_Test"."4UZ2".Ack OR "Data_base".xReset,
                   SimMode := "DB_Drives_Test".Sim_On,
                   HWID_Tel220 := "Drive_unit_1~PROFINET_interface~4UZ2_SIEMENS_telegram_220",
                   SpeedSp := "DB_Crane_Control".qr_Drive_SpeedSetpoint,
                   TorqueLimit := 100.0,
                   QuickStop := "DB_Crane_Control".qx_Drive_QuickStop,
                   CoastStop := "DB_Drives_Test"."4UZ2".CoastStop,
                   BrakesReleased := FALSE);
END_REGION
END_FUNCTION

FUNCTION "FC_Drives_HMI" : Void   // FC51, LAD
{ S7_Optimized_Access := 'TRUE' }
VERSION : 0.1
BEGIN

REGION Network 2 (SCL): Копіювання даних ПЧ 1UZ1 на візуалізацію
   // ============================================================
   // 1. Основні значення та діагностика драйвера
   // ============================================================

   "HMI_DB".Drives.Drive_1UZ1.Values.AxisEnabled := "DB_Drive_1UZ1".AxisEnabled;
   "HMI_DB".Drives.Drive_1UZ1.Values.Lockout := "DB_Drive_1UZ1".Lockout;
   "HMI_DB".Drives.Drive_1UZ1.Values.Error := "DB_Drive_1UZ1".Error;
   "HMI_DB".Drives.Drive_1UZ1.Values.BrakeOpenRequest := "DB_Drive_1UZ1".BrakeOpenRequest;

   "HMI_DB".Drives.Drive_1UZ1.Values.ActVelocity_Rpm := "DB_Drive_1UZ1".ActVelocity;
   "HMI_DB".Drives.Drive_1UZ1.Values.SpeedSetpointFb_Rpm := "DB_Drive_1UZ1".SpeedSetpointFb;
   "HMI_DB".Drives.Drive_1UZ1.Values.ActCurrent_A := "DB_Drive_1UZ1".ActCurrent;
   "HMI_DB".Drives.Drive_1UZ1.Values.ActTorque_Nm := "DB_Drive_1UZ1".ActTorque;
   "HMI_DB".Drives.Drive_1UZ1.Values.ActPower_kW := "DB_Drive_1UZ1".ActPower;
   "HMI_DB".Drives.Drive_1UZ1.Values.LoadPower_Pct := "DB_Drive_1UZ1".LoadPower;

   "HMI_DB".Drives.Drive_1UZ1.Values.FaultCode := "DB_Drive_1UZ1".FaultCode;
   "HMI_DB".Drives.Drive_1UZ1.Values.WarningCode := "DB_Drive_1UZ1".WarningCode;
   "HMI_DB".Drives.Drive_1UZ1.Values.Status := "DB_Drive_1UZ1".Status;
   "HMI_DB".Drives.Drive_1UZ1.Values.DiagId := "DB_Drive_1UZ1".DiagId;

   "HMI_DB".Drives.Drive_1UZ1.Values.SpeedError_Rpm := "DB_Drive_1UZ1".SpeedSetpointFb - "DB_Drive_1UZ1".ActVelocity;

   // ============================================================
   // Status driver bits
   // ============================================================

   "HMI_DB".Drives.Drive_1UZ1.StatusBits.ReadOk := "DB_Drive_1UZ1".Status.%X0;
   "HMI_DB".Drives.Drive_1UZ1.StatusBits.WriteOk := "DB_Drive_1UZ1".Status.%X1;
   "HMI_DB".Drives.Drive_1UZ1.StatusBits.AxisEnabled := "DB_Drive_1UZ1".Status.%X2;
   "HMI_DB".Drives.Drive_1UZ1.StatusBits.Lockout := "DB_Drive_1UZ1".Status.%X3;
   "HMI_DB".Drives.Drive_1UZ1.StatusBits.DriveFault := "DB_Drive_1UZ1".Status.%X4;
   "HMI_DB".Drives.Drive_1UZ1.StatusBits.DriveWarning := "DB_Drive_1UZ1".Status.%X5;
   "HMI_DB".Drives.Drive_1UZ1.StatusBits.BrakeOpenRequest := "DB_Drive_1UZ1".Status.%X6;
   "HMI_DB".Drives.Drive_1UZ1.StatusBits.SimMode := "DB_Drive_1UZ1".Status.%X7;
   "HMI_DB".Drives.Drive_1UZ1.StatusBits.SwitchingOnInhibit := "DB_Drive_1UZ1".Status.%X8;
   "HMI_DB".Drives.Drive_1UZ1.StatusBits.ControlRequested := "DB_Drive_1UZ1".Status.%X9;
   "HMI_DB".Drives.Drive_1UZ1.StatusBits.Reserved10 := "DB_Drive_1UZ1".Status.%X10;
   "HMI_DB".Drives.Drive_1UZ1.StatusBits.Reserved11 := "DB_Drive_1UZ1".Status.%X11;
   "HMI_DB".Drives.Drive_1UZ1.StatusBits.Reserved12 := "DB_Drive_1UZ1".Status.%X12;
   "HMI_DB".Drives.Drive_1UZ1.StatusBits.Reserved13 := "DB_Drive_1UZ1".Status.%X13;
   "HMI_DB".Drives.Drive_1UZ1.StatusBits.Reserved14 := "DB_Drive_1UZ1".Status.%X14;
   "HMI_DB".Drives.Drive_1UZ1.StatusBits.Reserved15 := "DB_Drive_1UZ1".Status.%X15;

   // ============================================================
   // 2. Raw telegram PLC -> ПЧ
   // ============================================================

   "HMI_DB".Drives.Drive_1UZ1.Raw.STW1_BM := "DB_Drive_1UZ1".TelOut.STW1_BM;
   "HMI_DB".Drives.Drive_1UZ1.Raw.NSOLL_B := "DB_Drive_1UZ1".TelOut.NSOLL_B;
   "HMI_DB".Drives.Drive_1UZ1.Raw.STW2_BM := "DB_Drive_1UZ1".TelOut.STW2_BM;
   "HMI_DB".Drives.Drive_1UZ1.Raw.M_ADD := "DB_Drive_1UZ1".TelOut.M_ADD;
   "HMI_DB".Drives.Drive_1UZ1.Raw.M_LIM := "DB_Drive_1UZ1".TelOut.M_LIM;
   "HMI_DB".Drives.Drive_1UZ1.Raw.USER_1 := "DB_Drive_1UZ1".TelOut.USER_1;
   "HMI_DB".Drives.Drive_1UZ1.Raw.USER_2 := "DB_Drive_1UZ1".TelOut.USER_2;
   "HMI_DB".Drives.Drive_1UZ1.Raw.USER_3 := "DB_Drive_1UZ1".TelOut.USER_3;
   "HMI_DB".Drives.Drive_1UZ1.Raw.USER_4 := "DB_Drive_1UZ1".TelOut.USER_4;



   // ============================================================
   // 3. Raw telegram ПЧ -> PLC
   // ============================================================

   "HMI_DB".Drives.Drive_1UZ1.Raw.ZSW1_BM := "DB_Drive_1UZ1".TelIn.ZSW1_BM;
   "HMI_DB".Drives.Drive_1UZ1.Raw.NIST_A := "DB_Drive_1UZ1".TelIn.NIST_A;
   "HMI_DB".Drives.Drive_1UZ1.Raw.IAIST := "DB_Drive_1UZ1".TelIn.IAIST;
   "HMI_DB".Drives.Drive_1UZ1.Raw.MIST := "DB_Drive_1UZ1".TelIn.MIST;
   "HMI_DB".Drives.Drive_1UZ1.Raw.WARN_CODE := "DB_Drive_1UZ1".TelIn.WARN_CODE;
   "HMI_DB".Drives.Drive_1UZ1.Raw.FAULT_CODE := "DB_Drive_1UZ1".TelIn.FAULT_CODE;
   "HMI_DB".Drives.Drive_1UZ1.Raw.ZSW2_BM := "DB_Drive_1UZ1".TelIn.ZSW2_BM;
   "HMI_DB".Drives.Drive_1UZ1.Raw.NSET_FB := "DB_Drive_1UZ1".TelIn.NSET_FB;
   "HMI_DB".Drives.Drive_1UZ1.Raw.P_ACT := "DB_Drive_1UZ1".TelIn.P_ACT;
   "HMI_DB".Drives.Drive_1UZ1.Raw.BRAKE_STATUS := "DB_Drive_1UZ1".TelIn.BRAKE_STATUS;


   // ============================================================
   // 4. STW1_BM bits, PLC -> ПЧ
   // ============================================================

   "HMI_DB".Drives.Drive_1UZ1.STW1.OnOff1 := "DB_Drive_1UZ1".TelOut.STW1_BM.%X0;
   "HMI_DB".Drives.Drive_1UZ1.STW1.NoCoastStop := "DB_Drive_1UZ1".TelOut.STW1_BM.%X1;
   "HMI_DB".Drives.Drive_1UZ1.STW1.NoQuickStop := "DB_Drive_1UZ1".TelOut.STW1_BM.%X2;
   "HMI_DB".Drives.Drive_1UZ1.STW1.EnableOperation := "DB_Drive_1UZ1".TelOut.STW1_BM.%X3;
   "HMI_DB".Drives.Drive_1UZ1.STW1.RampGeneratorEnable := "DB_Drive_1UZ1".TelOut.STW1_BM.%X4;
   "HMI_DB".Drives.Drive_1UZ1.STW1.RampGeneratorContinue := "DB_Drive_1UZ1".TelOut.STW1_BM.%X5;
   "HMI_DB".Drives.Drive_1UZ1.STW1.SetpointEnable := "DB_Drive_1UZ1".TelOut.STW1_BM.%X6;
   "HMI_DB".Drives.Drive_1UZ1.STW1.FaultAcknowledge := "DB_Drive_1UZ1".TelOut.STW1_BM.%X7;
   "HMI_DB".Drives.Drive_1UZ1.STW1.Reserved08 := "DB_Drive_1UZ1".TelOut.STW1_BM.%X8;
   "HMI_DB".Drives.Drive_1UZ1.STW1.Reserved09 := "DB_Drive_1UZ1".TelOut.STW1_BM.%X9;
   "HMI_DB".Drives.Drive_1UZ1.STW1.ControlByPLC := "DB_Drive_1UZ1".TelOut.STW1_BM.%X10;
   "HMI_DB".Drives.Drive_1UZ1.STW1.Reserved11 := "DB_Drive_1UZ1".TelOut.STW1_BM.%X11;
   "HMI_DB".Drives.Drive_1UZ1.STW1.Reserved12 := "DB_Drive_1UZ1".TelOut.STW1_BM.%X12;
   "HMI_DB".Drives.Drive_1UZ1.STW1.Reserved13 := "DB_Drive_1UZ1".TelOut.STW1_BM.%X13;
   "HMI_DB".Drives.Drive_1UZ1.STW1.Reserved14 := "DB_Drive_1UZ1".TelOut.STW1_BM.%X14;
   "HMI_DB".Drives.Drive_1UZ1.STW1.Reserved15 := "DB_Drive_1UZ1".TelOut.STW1_BM.%X15;


   // ============================================================
   // 5. STW2_BM bits, PLC -> ПЧ
   // ============================================================

   "HMI_DB".Drives.Drive_1UZ1.STW2.Bit00 := "DB_Drive_1UZ1".TelOut.STW2_BM.%X0;
   "HMI_DB".Drives.Drive_1UZ1.STW2.Bit01 := "DB_Drive_1UZ1".TelOut.STW2_BM.%X1;
   "HMI_DB".Drives.Drive_1UZ1.STW2.Bit02 := "DB_Drive_1UZ1".TelOut.STW2_BM.%X2;
   "HMI_DB".Drives.Drive_1UZ1.STW2.Bit03 := "DB_Drive_1UZ1".TelOut.STW2_BM.%X3;
   "HMI_DB".Drives.Drive_1UZ1.STW2.Bit04 := "DB_Drive_1UZ1".TelOut.STW2_BM.%X4;
   "HMI_DB".Drives.Drive_1UZ1.STW2.Bit05 := "DB_Drive_1UZ1".TelOut.STW2_BM.%X5;
   "HMI_DB".Drives.Drive_1UZ1.STW2.Bit06 := "DB_Drive_1UZ1".TelOut.STW2_BM.%X6;
   "HMI_DB".Drives.Drive_1UZ1.STW2.Bit07 := "DB_Drive_1UZ1".TelOut.STW2_BM.%X7;
   "HMI_DB".Drives.Drive_1UZ1.STW2.Bit08 := "DB_Drive_1UZ1".TelOut.STW2_BM.%X8;
   "HMI_DB".Drives.Drive_1UZ1.STW2.Bit09 := "DB_Drive_1UZ1".TelOut.STW2_BM.%X9;
   "HMI_DB".Drives.Drive_1UZ1.STW2.Bit10 := "DB_Drive_1UZ1".TelOut.STW2_BM.%X10;
   "HMI_DB".Drives.Drive_1UZ1.STW2.Bit11 := "DB_Drive_1UZ1".TelOut.STW2_BM.%X11;
   "HMI_DB".Drives.Drive_1UZ1.STW2.Bit12 := "DB_Drive_1UZ1".TelOut.STW2_BM.%X12;
   "HMI_DB".Drives.Drive_1UZ1.STW2.Bit13 := "DB_Drive_1UZ1".TelOut.STW2_BM.%X13;
   "HMI_DB".Drives.Drive_1UZ1.STW2.Bit14 := "DB_Drive_1UZ1".TelOut.STW2_BM.%X14;
   "HMI_DB".Drives.Drive_1UZ1.STW2.Bit15 := "DB_Drive_1UZ1".TelOut.STW2_BM.%X15;


   // ============================================================
   // 6. ZSW1_BM bits, ПЧ -> PLC
   // ============================================================

   "HMI_DB".Drives.Drive_1UZ1.ZSW1.ReadyToSwitchOn := "DB_Drive_1UZ1".TelIn.ZSW1_BM.%X0;
   "HMI_DB".Drives.Drive_1UZ1.ZSW1.ReadyToOperate := "DB_Drive_1UZ1".TelIn.ZSW1_BM.%X1;
   "HMI_DB".Drives.Drive_1UZ1.ZSW1.OperationEnabled := "DB_Drive_1UZ1".TelIn.ZSW1_BM.%X2;
   "HMI_DB".Drives.Drive_1UZ1.ZSW1.FaultActive := "DB_Drive_1UZ1".TelIn.ZSW1_BM.%X3;
   "HMI_DB".Drives.Drive_1UZ1.ZSW1.NoCoastStopActive := "DB_Drive_1UZ1".TelIn.ZSW1_BM.%X4;
   "HMI_DB".Drives.Drive_1UZ1.ZSW1.NoQuickStopActive := "DB_Drive_1UZ1".TelIn.ZSW1_BM.%X5;
   "HMI_DB".Drives.Drive_1UZ1.ZSW1.SwitchingOnInhibit := "DB_Drive_1UZ1".TelIn.ZSW1_BM.%X6;
   "HMI_DB".Drives.Drive_1UZ1.ZSW1.WarningActive := "DB_Drive_1UZ1".TelIn.ZSW1_BM.%X7;
   "HMI_DB".Drives.Drive_1UZ1.ZSW1.SpeedErrorInTolerance := "DB_Drive_1UZ1".TelIn.ZSW1_BM.%X8;
   "HMI_DB".Drives.Drive_1UZ1.ZSW1.ControlRequested := "DB_Drive_1UZ1".TelIn.ZSW1_BM.%X9;
   "HMI_DB".Drives.Drive_1UZ1.ZSW1.SetpointReached := "DB_Drive_1UZ1".TelIn.ZSW1_BM.%X10;
   "HMI_DB".Drives.Drive_1UZ1.ZSW1.InternalLimitActive := "DB_Drive_1UZ1".TelIn.ZSW1_BM.%X11;
   "HMI_DB".Drives.Drive_1UZ1.ZSW1.Reserved12 := "DB_Drive_1UZ1".TelIn.ZSW1_BM.%X12;
   "HMI_DB".Drives.Drive_1UZ1.ZSW1.Reserved13 := "DB_Drive_1UZ1".TelIn.ZSW1_BM.%X13;
   "HMI_DB".Drives.Drive_1UZ1.ZSW1.Reserved14 := "DB_Drive_1UZ1".TelIn.ZSW1_BM.%X14;
   "HMI_DB".Drives.Drive_1UZ1.ZSW1.Reserved15 := "DB_Drive_1UZ1".TelIn.ZSW1_BM.%X15;


   // ============================================================
   // 7. ZSW2_BM bits, ПЧ -> PLC
   // ============================================================

   "HMI_DB".Drives.Drive_1UZ1.ZSW2.Bit00 := "DB_Drive_1UZ1".TelIn.ZSW2_BM.%X0;
   "HMI_DB".Drives.Drive_1UZ1.ZSW2.Bit01 := "DB_Drive_1UZ1".TelIn.ZSW2_BM.%X1;
   "HMI_DB".Drives.Drive_1UZ1.ZSW2.Bit02 := "DB_Drive_1UZ1".TelIn.ZSW2_BM.%X2;
   "HMI_DB".Drives.Drive_1UZ1.ZSW2.Bit03 := "DB_Drive_1UZ1".TelIn.ZSW2_BM.%X3;
   "HMI_DB".Drives.Drive_1UZ1.ZSW2.Bit04 := "DB_Drive_1UZ1".TelIn.ZSW2_BM.%X4;
   "HMI_DB".Drives.Drive_1UZ1.ZSW2.Bit05 := "DB_Drive_1UZ1".TelIn.ZSW2_BM.%X5;
   "HMI_DB".Drives.Drive_1UZ1.ZSW2.Bit06 := "DB_Drive_1UZ1".TelIn.ZSW2_BM.%X6;
   "HMI_DB".Drives.Drive_1UZ1.ZSW2.Bit07 := "DB_Drive_1UZ1".TelIn.ZSW2_BM.%X7;
   "HMI_DB".Drives.Drive_1UZ1.ZSW2.Bit08 := "DB_Drive_1UZ1".TelIn.ZSW2_BM.%X8;
   "HMI_DB".Drives.Drive_1UZ1.ZSW2.Bit09 := "DB_Drive_1UZ1".TelIn.ZSW2_BM.%X9;
   "HMI_DB".Drives.Drive_1UZ1.ZSW2.Bit10 := "DB_Drive_1UZ1".TelIn.ZSW2_BM.%X10;
   "HMI_DB".Drives.Drive_1UZ1.ZSW2.Bit11 := "DB_Drive_1UZ1".TelIn.ZSW2_BM.%X11;
   "HMI_DB".Drives.Drive_1UZ1.ZSW2.Bit12 := "DB_Drive_1UZ1".TelIn.ZSW2_BM.%X12;
   "HMI_DB".Drives.Drive_1UZ1.ZSW2.Bit13 := "DB_Drive_1UZ1".TelIn.ZSW2_BM.%X13;
   "HMI_DB".Drives.Drive_1UZ1.ZSW2.Bit14 := "DB_Drive_1UZ1".TelIn.ZSW2_BM.%X14;
   "HMI_DB".Drives.Drive_1UZ1.ZSW2.Bit15 := "DB_Drive_1UZ1".TelIn.ZSW2_BM.%X15;


   // ============================================================
   // 8. BRAKE_STATUS / r1229 bits, ПЧ -> PLC
   // ============================================================

   "HMI_DB".Drives.Drive_1UZ1.Brake.RawWord := "DB_Drive_1UZ1".TelIn.BRAKE_STATUS;

   "HMI_DB".Drives.Drive_1UZ1.Brake.Bit00 := "DB_Drive_1UZ1".TelIn.BRAKE_STATUS.%X0;
   "HMI_DB".Drives.Drive_1UZ1.Brake.CommandOpenBrake := "DB_Drive_1UZ1".TelIn.BRAKE_STATUS.%X1;
   "HMI_DB".Drives.Drive_1UZ1.Brake.Bit02 := "DB_Drive_1UZ1".TelIn.BRAKE_STATUS.%X2;
   "HMI_DB".Drives.Drive_1UZ1.Brake.PulseEnableExtendedBrakeControl := "DB_Drive_1UZ1".TelIn.BRAKE_STATUS.%X3;
   "HMI_DB".Drives.Drive_1UZ1.Brake.BrakeDoesNotOpen := "DB_Drive_1UZ1".TelIn.BRAKE_STATUS.%X4;
   "HMI_DB".Drives.Drive_1UZ1.Brake.BrakeDoesNotClose := "DB_Drive_1UZ1".TelIn.BRAKE_STATUS.%X5;
   "HMI_DB".Drives.Drive_1UZ1.Brake.BrakeThresholdExceeded := "DB_Drive_1UZ1".TelIn.BRAKE_STATUS.%X6;
   "HMI_DB".Drives.Drive_1UZ1.Brake.BrakeThresholdUndershot := "DB_Drive_1UZ1".TelIn.BRAKE_STATUS.%X7;
   "HMI_DB".Drives.Drive_1UZ1.Brake.BrakeMonitoringTimeExpired := "DB_Drive_1UZ1".TelIn.BRAKE_STATUS.%X8;
   "HMI_DB".Drives.Drive_1UZ1.Brake.PulseEnableRequestMissing := "DB_Drive_1UZ1".TelIn.BRAKE_STATUS.%X9;
   "HMI_DB".Drives.Drive_1UZ1.Brake.BrakeOrLogicResult := "DB_Drive_1UZ1".TelIn.BRAKE_STATUS.%X10;
   "HMI_DB".Drives.Drive_1UZ1.Brake.BrakeAndLogicResult := "DB_Drive_1UZ1".TelIn.BRAKE_STATUS.%X11;
   "HMI_DB".Drives.Drive_1UZ1.Brake.Bit12 := "DB_Drive_1UZ1".TelIn.BRAKE_STATUS.%X12;
   "HMI_DB".Drives.Drive_1UZ1.Brake.Bit13 := "DB_Drive_1UZ1".TelIn.BRAKE_STATUS.%X13;
   "HMI_DB".Drives.Drive_1UZ1.Brake.Bit14 := "DB_Drive_1UZ1".TelIn.BRAKE_STATUS.%X14;
   "HMI_DB".Drives.Drive_1UZ1.Brake.Bit15 := "DB_Drive_1UZ1".TelIn.BRAKE_STATUS.%X15;
END_REGION

REGION Network 3 (SCL): Копіювання даних ПЧ 3UZ1 на візуалізацію
   // ============================================================
   // 1. Основні значення та діагностика драйвера
   // ============================================================

   "HMI_DB".Drives.Drive_3UZ1.Values.AxisEnabled := "DB_Drive_3UZ1".AxisEnabled;
   "HMI_DB".Drives.Drive_3UZ1.Values.Lockout := "DB_Drive_3UZ1".Lockout;
   "HMI_DB".Drives.Drive_3UZ1.Values.Error := "DB_Drive_3UZ1".Error;
   "HMI_DB".Drives.Drive_3UZ1.Values.BrakeOpenRequest := "DB_Drive_3UZ1".BrakeOpenRequest;

   "HMI_DB".Drives.Drive_3UZ1.Values.ActVelocity_Rpm := "DB_Drive_3UZ1".ActVelocity;
   "HMI_DB".Drives.Drive_3UZ1.Values.SpeedSetpointFb_Rpm := "DB_Drive_3UZ1".SpeedSetpointFb;
   "HMI_DB".Drives.Drive_3UZ1.Values.ActCurrent_A := "DB_Drive_3UZ1".ActCurrent;
   "HMI_DB".Drives.Drive_3UZ1.Values.ActTorque_Nm := "DB_Drive_3UZ1".ActTorque;
   "HMI_DB".Drives.Drive_3UZ1.Values.ActPower_kW := "DB_Drive_3UZ1".ActPower;
   "HMI_DB".Drives.Drive_3UZ1.Values.LoadPower_Pct := "DB_Drive_3UZ1".LoadPower;

   "HMI_DB".Drives.Drive_3UZ1.Values.FaultCode := "DB_Drive_3UZ1".FaultCode;
   "HMI_DB".Drives.Drive_3UZ1.Values.WarningCode := "DB_Drive_3UZ1".WarningCode;
   "HMI_DB".Drives.Drive_3UZ1.Values.Status := "DB_Drive_3UZ1".Status;
   "HMI_DB".Drives.Drive_3UZ1.Values.DiagId := "DB_Drive_3UZ1".DiagId;

   "HMI_DB".Drives.Drive_3UZ1.Values.SpeedError_Rpm := "DB_Drive_3UZ1".SpeedSetpointFb - "DB_Drive_3UZ1".ActVelocity;

   // ============================================================
   // Status driver bits
   // ============================================================

   "HMI_DB".Drives.Drive_3UZ1.StatusBits.ReadOk := "DB_Drive_3UZ1".Status.%X0;
   "HMI_DB".Drives.Drive_3UZ1.StatusBits.WriteOk := "DB_Drive_3UZ1".Status.%X1;
   "HMI_DB".Drives.Drive_3UZ1.StatusBits.AxisEnabled := "DB_Drive_3UZ1".Status.%X2;
   "HMI_DB".Drives.Drive_3UZ1.StatusBits.Lockout := "DB_Drive_3UZ1".Status.%X3;
   "HMI_DB".Drives.Drive_3UZ1.StatusBits.DriveFault := "DB_Drive_3UZ1".Status.%X4;
   "HMI_DB".Drives.Drive_3UZ1.StatusBits.DriveWarning := "DB_Drive_3UZ1".Status.%X5;
   "HMI_DB".Drives.Drive_3UZ1.StatusBits.BrakeOpenRequest := "DB_Drive_3UZ1".Status.%X6;
   "HMI_DB".Drives.Drive_3UZ1.StatusBits.SimMode := "DB_Drive_3UZ1".Status.%X7;
   "HMI_DB".Drives.Drive_3UZ1.StatusBits.SwitchingOnInhibit := "DB_Drive_3UZ1".Status.%X8;
   "HMI_DB".Drives.Drive_3UZ1.StatusBits.ControlRequested := "DB_Drive_3UZ1".Status.%X9;
   "HMI_DB".Drives.Drive_3UZ1.StatusBits.Reserved10 := "DB_Drive_3UZ1".Status.%X10;
   "HMI_DB".Drives.Drive_3UZ1.StatusBits.Reserved11 := "DB_Drive_3UZ1".Status.%X11;
   "HMI_DB".Drives.Drive_3UZ1.StatusBits.Reserved12 := "DB_Drive_3UZ1".Status.%X12;
   "HMI_DB".Drives.Drive_3UZ1.StatusBits.Reserved13 := "DB_Drive_3UZ1".Status.%X13;
   "HMI_DB".Drives.Drive_3UZ1.StatusBits.Reserved14 := "DB_Drive_3UZ1".Status.%X14;
   "HMI_DB".Drives.Drive_3UZ1.StatusBits.Reserved15 := "DB_Drive_3UZ1".Status.%X15;

   // ============================================================
   // 2. Raw telegram PLC -> ПЧ
   // ============================================================

   "HMI_DB".Drives.Drive_3UZ1.Raw.STW1_BM := "DB_Drive_3UZ1".TelOut.STW1_BM;
   "HMI_DB".Drives.Drive_3UZ1.Raw.NSOLL_B := "DB_Drive_3UZ1".TelOut.NSOLL_B;
   "HMI_DB".Drives.Drive_3UZ1.Raw.STW2_BM := "DB_Drive_3UZ1".TelOut.STW2_BM;
   "HMI_DB".Drives.Drive_3UZ1.Raw.M_ADD := "DB_Drive_3UZ1".TelOut.M_ADD;
   "HMI_DB".Drives.Drive_3UZ1.Raw.M_LIM := "DB_Drive_3UZ1".TelOut.M_LIM;
   "HMI_DB".Drives.Drive_3UZ1.Raw.USER_1 := "DB_Drive_3UZ1".TelOut.USER_1;
   "HMI_DB".Drives.Drive_3UZ1.Raw.USER_2 := "DB_Drive_3UZ1".TelOut.USER_2;
   "HMI_DB".Drives.Drive_3UZ1.Raw.USER_3 := "DB_Drive_3UZ1".TelOut.USER_3;
   "HMI_DB".Drives.Drive_3UZ1.Raw.USER_4 := "DB_Drive_3UZ1".TelOut.USER_4;



   // ============================================================
   // 3. Raw telegram ПЧ -> PLC
   // ============================================================

   "HMI_DB".Drives.Drive_3UZ1.Raw.ZSW1_BM := "DB_Drive_3UZ1".TelIn.ZSW1_BM;
   "HMI_DB".Drives.Drive_3UZ1.Raw.NIST_A := "DB_Drive_3UZ1".TelIn.NIST_A;
   "HMI_DB".Drives.Drive_3UZ1.Raw.IAIST := "DB_Drive_3UZ1".TelIn.IAIST;
   "HMI_DB".Drives.Drive_3UZ1.Raw.MIST := "DB_Drive_3UZ1".TelIn.MIST;
   "HMI_DB".Drives.Drive_3UZ1.Raw.WARN_CODE := "DB_Drive_3UZ1".TelIn.WARN_CODE;
   "HMI_DB".Drives.Drive_3UZ1.Raw.FAULT_CODE := "DB_Drive_3UZ1".TelIn.FAULT_CODE;
   "HMI_DB".Drives.Drive_3UZ1.Raw.ZSW2_BM := "DB_Drive_3UZ1".TelIn.ZSW2_BM;
   "HMI_DB".Drives.Drive_3UZ1.Raw.NSET_FB := "DB_Drive_3UZ1".TelIn.NSET_FB;
   "HMI_DB".Drives.Drive_3UZ1.Raw.P_ACT := "DB_Drive_3UZ1".TelIn.P_ACT;
   "HMI_DB".Drives.Drive_3UZ1.Raw.BRAKE_STATUS := "DB_Drive_3UZ1".TelIn.BRAKE_STATUS;


   // ============================================================
   // 4. STW1_BM bits, PLC -> ПЧ
   // ============================================================

   "HMI_DB".Drives.Drive_3UZ1.STW1.OnOff1 := "DB_Drive_3UZ1".TelOut.STW1_BM.%X0;
   "HMI_DB".Drives.Drive_3UZ1.STW1.NoCoastStop := "DB_Drive_3UZ1".TelOut.STW1_BM.%X1;
   "HMI_DB".Drives.Drive_3UZ1.STW1.NoQuickStop := "DB_Drive_3UZ1".TelOut.STW1_BM.%X2;
   "HMI_DB".Drives.Drive_3UZ1.STW1.EnableOperation := "DB_Drive_3UZ1".TelOut.STW1_BM.%X3;
   "HMI_DB".Drives.Drive_3UZ1.STW1.RampGeneratorEnable := "DB_Drive_3UZ1".TelOut.STW1_BM.%X4;
   "HMI_DB".Drives.Drive_3UZ1.STW1.RampGeneratorContinue := "DB_Drive_3UZ1".TelOut.STW1_BM.%X5;
   "HMI_DB".Drives.Drive_3UZ1.STW1.SetpointEnable := "DB_Drive_3UZ1".TelOut.STW1_BM.%X6;
   "HMI_DB".Drives.Drive_3UZ1.STW1.FaultAcknowledge := "DB_Drive_3UZ1".TelOut.STW1_BM.%X7;
   "HMI_DB".Drives.Drive_3UZ1.STW1.Reserved08 := "DB_Drive_3UZ1".TelOut.STW1_BM.%X8;
   "HMI_DB".Drives.Drive_3UZ1.STW1.Reserved09 := "DB_Drive_3UZ1".TelOut.STW1_BM.%X9;
   "HMI_DB".Drives.Drive_3UZ1.STW1.ControlByPLC := "DB_Drive_3UZ1".TelOut.STW1_BM.%X10;
   "HMI_DB".Drives.Drive_3UZ1.STW1.Reserved11 := "DB_Drive_3UZ1".TelOut.STW1_BM.%X11;
   "HMI_DB".Drives.Drive_3UZ1.STW1.Reserved12 := "DB_Drive_3UZ1".TelOut.STW1_BM.%X12;
   "HMI_DB".Drives.Drive_3UZ1.STW1.Reserved13 := "DB_Drive_3UZ1".TelOut.STW1_BM.%X13;
   "HMI_DB".Drives.Drive_3UZ1.STW1.Reserved14 := "DB_Drive_3UZ1".TelOut.STW1_BM.%X14;
   "HMI_DB".Drives.Drive_3UZ1.STW1.Reserved15 := "DB_Drive_3UZ1".TelOut.STW1_BM.%X15;


   // ============================================================
   // 5. STW2_BM bits, PLC -> ПЧ
   // ============================================================

   "HMI_DB".Drives.Drive_3UZ1.STW2.Bit00 := "DB_Drive_3UZ1".TelOut.STW2_BM.%X0;
   "HMI_DB".Drives.Drive_3UZ1.STW2.Bit01 := "DB_Drive_3UZ1".TelOut.STW2_BM.%X1;
   "HMI_DB".Drives.Drive_3UZ1.STW2.Bit02 := "DB_Drive_3UZ1".TelOut.STW2_BM.%X2;
   "HMI_DB".Drives.Drive_3UZ1.STW2.Bit03 := "DB_Drive_3UZ1".TelOut.STW2_BM.%X3;
   "HMI_DB".Drives.Drive_3UZ1.STW2.Bit04 := "DB_Drive_3UZ1".TelOut.STW2_BM.%X4;
   "HMI_DB".Drives.Drive_3UZ1.STW2.Bit05 := "DB_Drive_3UZ1".TelOut.STW2_BM.%X5;
   "HMI_DB".Drives.Drive_3UZ1.STW2.Bit06 := "DB_Drive_3UZ1".TelOut.STW2_BM.%X6;
   "HMI_DB".Drives.Drive_3UZ1.STW2.Bit07 := "DB_Drive_3UZ1".TelOut.STW2_BM.%X7;
   "HMI_DB".Drives.Drive_3UZ1.STW2.Bit08 := "DB_Drive_3UZ1".TelOut.STW2_BM.%X8;
   "HMI_DB".Drives.Drive_3UZ1.STW2.Bit09 := "DB_Drive_3UZ1".TelOut.STW2_BM.%X9;
   "HMI_DB".Drives.Drive_3UZ1.STW2.Bit10 := "DB_Drive_3UZ1".TelOut.STW2_BM.%X10;
   "HMI_DB".Drives.Drive_3UZ1.STW2.Bit11 := "DB_Drive_3UZ1".TelOut.STW2_BM.%X11;
   "HMI_DB".Drives.Drive_3UZ1.STW2.Bit12 := "DB_Drive_3UZ1".TelOut.STW2_BM.%X12;
   "HMI_DB".Drives.Drive_3UZ1.STW2.Bit13 := "DB_Drive_3UZ1".TelOut.STW2_BM.%X13;
   "HMI_DB".Drives.Drive_3UZ1.STW2.Bit14 := "DB_Drive_3UZ1".TelOut.STW2_BM.%X14;
   "HMI_DB".Drives.Drive_3UZ1.STW2.Bit15 := "DB_Drive_3UZ1".TelOut.STW2_BM.%X15;


   // ============================================================
   // 6. ZSW1_BM bits, ПЧ -> PLC
   // ============================================================

   "HMI_DB".Drives.Drive_3UZ1.ZSW1.ReadyToSwitchOn := "DB_Drive_3UZ1".TelIn.ZSW1_BM.%X0;
   "HMI_DB".Drives.Drive_3UZ1.ZSW1.ReadyToOperate := "DB_Drive_3UZ1".TelIn.ZSW1_BM.%X1;
   "HMI_DB".Drives.Drive_3UZ1.ZSW1.OperationEnabled := "DB_Drive_3UZ1".TelIn.ZSW1_BM.%X2;
   "HMI_DB".Drives.Drive_3UZ1.ZSW1.FaultActive := "DB_Drive_3UZ1".TelIn.ZSW1_BM.%X3;
   "HMI_DB".Drives.Drive_3UZ1.ZSW1.NoCoastStopActive := "DB_Drive_3UZ1".TelIn.ZSW1_BM.%X4;
   "HMI_DB".Drives.Drive_3UZ1.ZSW1.NoQuickStopActive := "DB_Drive_3UZ1".TelIn.ZSW1_BM.%X5;
   "HMI_DB".Drives.Drive_3UZ1.ZSW1.SwitchingOnInhibit := "DB_Drive_3UZ1".TelIn.ZSW1_BM.%X6;
   "HMI_DB".Drives.Drive_3UZ1.ZSW1.WarningActive := "DB_Drive_3UZ1".TelIn.ZSW1_BM.%X7;
   "HMI_DB".Drives.Drive_3UZ1.ZSW1.SpeedErrorInTolerance := "DB_Drive_3UZ1".TelIn.ZSW1_BM.%X8;
   "HMI_DB".Drives.Drive_3UZ1.ZSW1.ControlRequested := "DB_Drive_3UZ1".TelIn.ZSW1_BM.%X9;
   "HMI_DB".Drives.Drive_3UZ1.ZSW1.SetpointReached := "DB_Drive_3UZ1".TelIn.ZSW1_BM.%X10;
   "HMI_DB".Drives.Drive_3UZ1.ZSW1.InternalLimitActive := "DB_Drive_3UZ1".TelIn.ZSW1_BM.%X11;
   "HMI_DB".Drives.Drive_3UZ1.ZSW1.Reserved12 := "DB_Drive_3UZ1".TelIn.ZSW1_BM.%X12;
   "HMI_DB".Drives.Drive_3UZ1.ZSW1.Reserved13 := "DB_Drive_3UZ1".TelIn.ZSW1_BM.%X13;
   "HMI_DB".Drives.Drive_3UZ1.ZSW1.Reserved14 := "DB_Drive_3UZ1".TelIn.ZSW1_BM.%X14;
   "HMI_DB".Drives.Drive_3UZ1.ZSW1.Reserved15 := "DB_Drive_3UZ1".TelIn.ZSW1_BM.%X15;


   // ============================================================
   // 7. ZSW2_BM bits, ПЧ -> PLC
   // ============================================================

   "HMI_DB".Drives.Drive_3UZ1.ZSW2.Bit00 := "DB_Drive_3UZ1".TelIn.ZSW2_BM.%X0;
   "HMI_DB".Drives.Drive_3UZ1.ZSW2.Bit01 := "DB_Drive_3UZ1".TelIn.ZSW2_BM.%X1;
   "HMI_DB".Drives.Drive_3UZ1.ZSW2.Bit02 := "DB_Drive_3UZ1".TelIn.ZSW2_BM.%X2;
   "HMI_DB".Drives.Drive_3UZ1.ZSW2.Bit03 := "DB_Drive_3UZ1".TelIn.ZSW2_BM.%X3;
   "HMI_DB".Drives.Drive_3UZ1.ZSW2.Bit04 := "DB_Drive_3UZ1".TelIn.ZSW2_BM.%X4;
   "HMI_DB".Drives.Drive_3UZ1.ZSW2.Bit05 := "DB_Drive_3UZ1".TelIn.ZSW2_BM.%X5;
   "HMI_DB".Drives.Drive_3UZ1.ZSW2.Bit06 := "DB_Drive_3UZ1".TelIn.ZSW2_BM.%X6;
   "HMI_DB".Drives.Drive_3UZ1.ZSW2.Bit07 := "DB_Drive_3UZ1".TelIn.ZSW2_BM.%X7;
   "HMI_DB".Drives.Drive_3UZ1.ZSW2.Bit08 := "DB_Drive_3UZ1".TelIn.ZSW2_BM.%X8;
   "HMI_DB".Drives.Drive_3UZ1.ZSW2.Bit09 := "DB_Drive_3UZ1".TelIn.ZSW2_BM.%X9;
   "HMI_DB".Drives.Drive_3UZ1.ZSW2.Bit10 := "DB_Drive_3UZ1".TelIn.ZSW2_BM.%X10;
   "HMI_DB".Drives.Drive_3UZ1.ZSW2.Bit11 := "DB_Drive_3UZ1".TelIn.ZSW2_BM.%X11;
   "HMI_DB".Drives.Drive_3UZ1.ZSW2.Bit12 := "DB_Drive_3UZ1".TelIn.ZSW2_BM.%X12;
   "HMI_DB".Drives.Drive_3UZ1.ZSW2.Bit13 := "DB_Drive_3UZ1".TelIn.ZSW2_BM.%X13;
   "HMI_DB".Drives.Drive_3UZ1.ZSW2.Bit14 := "DB_Drive_3UZ1".TelIn.ZSW2_BM.%X14;
   "HMI_DB".Drives.Drive_3UZ1.ZSW2.Bit15 := "DB_Drive_3UZ1".TelIn.ZSW2_BM.%X15;


   // ============================================================
   // 8. BRAKE_STATUS / r1229 bits, ПЧ -> PLC
   // ============================================================

   "HMI_DB".Drives.Drive_3UZ1.Brake.RawWord := "DB_Drive_3UZ1".TelIn.BRAKE_STATUS;

   "HMI_DB".Drives.Drive_3UZ1.Brake.Bit00 := "DB_Drive_3UZ1".TelIn.BRAKE_STATUS.%X0;
   "HMI_DB".Drives.Drive_3UZ1.Brake.CommandOpenBrake := "DB_Drive_3UZ1".TelIn.BRAKE_STATUS.%X1;
   "HMI_DB".Drives.Drive_3UZ1.Brake.Bit02 := "DB_Drive_3UZ1".TelIn.BRAKE_STATUS.%X2;
   "HMI_DB".Drives.Drive_3UZ1.Brake.PulseEnableExtendedBrakeControl := "DB_Drive_3UZ1".TelIn.BRAKE_STATUS.%X3;
   "HMI_DB".Drives.Drive_3UZ1.Brake.BrakeDoesNotOpen := "DB_Drive_3UZ1".TelIn.BRAKE_STATUS.%X4;
   "HMI_DB".Drives.Drive_3UZ1.Brake.BrakeDoesNotClose := "DB_Drive_3UZ1".TelIn.BRAKE_STATUS.%X5;
   "HMI_DB".Drives.Drive_3UZ1.Brake.BrakeThresholdExceeded := "DB_Drive_3UZ1".TelIn.BRAKE_STATUS.%X6;
   "HMI_DB".Drives.Drive_3UZ1.Brake.BrakeThresholdUndershot := "DB_Drive_3UZ1".TelIn.BRAKE_STATUS.%X7;
   "HMI_DB".Drives.Drive_3UZ1.Brake.BrakeMonitoringTimeExpired := "DB_Drive_3UZ1".TelIn.BRAKE_STATUS.%X8;
   "HMI_DB".Drives.Drive_3UZ1.Brake.PulseEnableRequestMissing := "DB_Drive_3UZ1".TelIn.BRAKE_STATUS.%X9;
   "HMI_DB".Drives.Drive_3UZ1.Brake.BrakeOrLogicResult := "DB_Drive_3UZ1".TelIn.BRAKE_STATUS.%X10;
   "HMI_DB".Drives.Drive_3UZ1.Brake.BrakeAndLogicResult := "DB_Drive_3UZ1".TelIn.BRAKE_STATUS.%X11;
   "HMI_DB".Drives.Drive_3UZ1.Brake.Bit12 := "DB_Drive_3UZ1".TelIn.BRAKE_STATUS.%X12;
   "HMI_DB".Drives.Drive_3UZ1.Brake.Bit13 := "DB_Drive_3UZ1".TelIn.BRAKE_STATUS.%X13;
   "HMI_DB".Drives.Drive_3UZ1.Brake.Bit14 := "DB_Drive_3UZ1".TelIn.BRAKE_STATUS.%X14;
   "HMI_DB".Drives.Drive_3UZ1.Brake.Bit15 := "DB_Drive_3UZ1".TelIn.BRAKE_STATUS.%X15;
END_REGION

REGION Network 4 (SCL): Копіювання даних ПЧ 4UZ1 на візуалізацію
   // ============================================================
   // 1. Основні значення та діагностика драйвера
   // ============================================================

   "HMI_DB".Drives.Drive_4UZ1.Values.AxisEnabled := "DB_Drive_4UZ1".AxisEnabled;
   "HMI_DB".Drives.Drive_4UZ1.Values.Lockout := "DB_Drive_4UZ1".Lockout;
   "HMI_DB".Drives.Drive_4UZ1.Values.Error := "DB_Drive_4UZ1".Error;
   "HMI_DB".Drives.Drive_4UZ1.Values.BrakeOpenRequest := "DB_Drive_4UZ1".BrakeOpenRequest;

   "HMI_DB".Drives.Drive_4UZ1.Values.ActVelocity_Rpm := "DB_Drive_4UZ1".ActVelocity;
   "HMI_DB".Drives.Drive_4UZ1.Values.SpeedSetpointFb_Rpm := "DB_Drive_4UZ1".SpeedSetpointFb;
   "HMI_DB".Drives.Drive_4UZ1.Values.ActCurrent_A := "DB_Drive_4UZ1".ActCurrent;
   "HMI_DB".Drives.Drive_4UZ1.Values.ActTorque_Nm := "DB_Drive_4UZ1".ActTorque;
   "HMI_DB".Drives.Drive_4UZ1.Values.ActPower_kW := "DB_Drive_4UZ1".ActPower;
   "HMI_DB".Drives.Drive_4UZ1.Values.LoadPower_Pct := "DB_Drive_4UZ1".LoadPower;

   "HMI_DB".Drives.Drive_4UZ1.Values.FaultCode := "DB_Drive_4UZ1".FaultCode;
   "HMI_DB".Drives.Drive_4UZ1.Values.WarningCode := "DB_Drive_4UZ1".WarningCode;
   "HMI_DB".Drives.Drive_4UZ1.Values.Status := "DB_Drive_4UZ1".Status;
   "HMI_DB".Drives.Drive_4UZ1.Values.DiagId := "DB_Drive_4UZ1".DiagId;

   "HMI_DB".Drives.Drive_4UZ1.Values.SpeedError_Rpm := "DB_Drive_4UZ1".SpeedSetpointFb - "DB_Drive_4UZ1".ActVelocity;

   // ============================================================
   // Status driver bits
   // ============================================================

   "HMI_DB".Drives.Drive_4UZ1.StatusBits.ReadOk := "DB_Drive_4UZ1".Status.%X0;
   "HMI_DB".Drives.Drive_4UZ1.StatusBits.WriteOk := "DB_Drive_4UZ1".Status.%X1;
   "HMI_DB".Drives.Drive_4UZ1.StatusBits.AxisEnabled := "DB_Drive_4UZ1".Status.%X2;
   "HMI_DB".Drives.Drive_4UZ1.StatusBits.Lockout := "DB_Drive_4UZ1".Status.%X3;
   "HMI_DB".Drives.Drive_4UZ1.StatusBits.DriveFault := "DB_Drive_4UZ1".Status.%X4;
   "HMI_DB".Drives.Drive_4UZ1.StatusBits.DriveWarning := "DB_Drive_4UZ1".Status.%X5;
   "HMI_DB".Drives.Drive_4UZ1.StatusBits.BrakeOpenRequest := "DB_Drive_4UZ1".Status.%X6;
   "HMI_DB".Drives.Drive_4UZ1.StatusBits.SimMode := "DB_Drive_4UZ1".Status.%X7;
   "HMI_DB".Drives.Drive_4UZ1.StatusBits.SwitchingOnInhibit := "DB_Drive_4UZ1".Status.%X8;
   "HMI_DB".Drives.Drive_4UZ1.StatusBits.ControlRequested := "DB_Drive_4UZ1".Status.%X9;
   "HMI_DB".Drives.Drive_4UZ1.StatusBits.Reserved10 := "DB_Drive_4UZ1".Status.%X10;
   "HMI_DB".Drives.Drive_4UZ1.StatusBits.Reserved11 := "DB_Drive_4UZ1".Status.%X11;
   "HMI_DB".Drives.Drive_4UZ1.StatusBits.Reserved12 := "DB_Drive_4UZ1".Status.%X12;
   "HMI_DB".Drives.Drive_4UZ1.StatusBits.Reserved13 := "DB_Drive_4UZ1".Status.%X13;
   "HMI_DB".Drives.Drive_4UZ1.StatusBits.Reserved14 := "DB_Drive_4UZ1".Status.%X14;
   "HMI_DB".Drives.Drive_4UZ1.StatusBits.Reserved15 := "DB_Drive_4UZ1".Status.%X15;

   // ============================================================
   // 2. Raw telegram PLC -> ПЧ
   // ============================================================

   "HMI_DB".Drives.Drive_4UZ1.Raw.STW1_BM := "DB_Drive_4UZ1".TelOut.STW1_BM;
   "HMI_DB".Drives.Drive_4UZ1.Raw.NSOLL_B := "DB_Drive_4UZ1".TelOut.NSOLL_B;
   "HMI_DB".Drives.Drive_4UZ1.Raw.STW2_BM := "DB_Drive_4UZ1".TelOut.STW2_BM;
   "HMI_DB".Drives.Drive_4UZ1.Raw.M_ADD := "DB_Drive_4UZ1".TelOut.M_ADD;
   "HMI_DB".Drives.Drive_4UZ1.Raw.M_LIM := "DB_Drive_4UZ1".TelOut.M_LIM;
   "HMI_DB".Drives.Drive_4UZ1.Raw.USER_1 := "DB_Drive_4UZ1".TelOut.USER_1;
   "HMI_DB".Drives.Drive_4UZ1.Raw.USER_2 := "DB_Drive_4UZ1".TelOut.USER_2;
   "HMI_DB".Drives.Drive_4UZ1.Raw.USER_3 := "DB_Drive_4UZ1".TelOut.USER_3;
   "HMI_DB".Drives.Drive_4UZ1.Raw.USER_4 := "DB_Drive_4UZ1".TelOut.USER_4;



   // ============================================================
   // 3. Raw telegram ПЧ -> PLC
   // ============================================================

   "HMI_DB".Drives.Drive_4UZ1.Raw.ZSW1_BM := "DB_Drive_4UZ1".TelIn.ZSW1_BM;
   "HMI_DB".Drives.Drive_4UZ1.Raw.NIST_A := "DB_Drive_4UZ1".TelIn.NIST_A;
   "HMI_DB".Drives.Drive_4UZ1.Raw.IAIST := "DB_Drive_4UZ1".TelIn.IAIST;
   "HMI_DB".Drives.Drive_4UZ1.Raw.MIST := "DB_Drive_4UZ1".TelIn.MIST;
   "HMI_DB".Drives.Drive_4UZ1.Raw.WARN_CODE := "DB_Drive_4UZ1".TelIn.WARN_CODE;
   "HMI_DB".Drives.Drive_4UZ1.Raw.FAULT_CODE := "DB_Drive_4UZ1".TelIn.FAULT_CODE;
   "HMI_DB".Drives.Drive_4UZ1.Raw.ZSW2_BM := "DB_Drive_4UZ1".TelIn.ZSW2_BM;
   "HMI_DB".Drives.Drive_4UZ1.Raw.NSET_FB := "DB_Drive_4UZ1".TelIn.NSET_FB;
   "HMI_DB".Drives.Drive_4UZ1.Raw.P_ACT := "DB_Drive_4UZ1".TelIn.P_ACT;
   "HMI_DB".Drives.Drive_4UZ1.Raw.BRAKE_STATUS := "DB_Drive_4UZ1".TelIn.BRAKE_STATUS;


   // ============================================================
   // 4. STW1_BM bits, PLC -> ПЧ
   // ============================================================

   "HMI_DB".Drives.Drive_4UZ1.STW1.OnOff1 := "DB_Drive_4UZ1".TelOut.STW1_BM.%X0;
   "HMI_DB".Drives.Drive_4UZ1.STW1.NoCoastStop := "DB_Drive_4UZ1".TelOut.STW1_BM.%X1;
   "HMI_DB".Drives.Drive_4UZ1.STW1.NoQuickStop := "DB_Drive_4UZ1".TelOut.STW1_BM.%X2;
   "HMI_DB".Drives.Drive_4UZ1.STW1.EnableOperation := "DB_Drive_4UZ1".TelOut.STW1_BM.%X3;
   "HMI_DB".Drives.Drive_4UZ1.STW1.RampGeneratorEnable := "DB_Drive_4UZ1".TelOut.STW1_BM.%X4;
   "HMI_DB".Drives.Drive_4UZ1.STW1.RampGeneratorContinue := "DB_Drive_4UZ1".TelOut.STW1_BM.%X5;
   "HMI_DB".Drives.Drive_4UZ1.STW1.SetpointEnable := "DB_Drive_4UZ1".TelOut.STW1_BM.%X6;
   "HMI_DB".Drives.Drive_4UZ1.STW1.FaultAcknowledge := "DB_Drive_4UZ1".TelOut.STW1_BM.%X7;
   "HMI_DB".Drives.Drive_4UZ1.STW1.Reserved08 := "DB_Drive_4UZ1".TelOut.STW1_BM.%X8;
   "HMI_DB".Drives.Drive_4UZ1.STW1.Reserved09 := "DB_Drive_4UZ1".TelOut.STW1_BM.%X9;
   "HMI_DB".Drives.Drive_4UZ1.STW1.ControlByPLC := "DB_Drive_4UZ1".TelOut.STW1_BM.%X10;
   "HMI_DB".Drives.Drive_4UZ1.STW1.Reserved11 := "DB_Drive_4UZ1".TelOut.STW1_BM.%X11;
   "HMI_DB".Drives.Drive_4UZ1.STW1.Reserved12 := "DB_Drive_4UZ1".TelOut.STW1_BM.%X12;
   "HMI_DB".Drives.Drive_4UZ1.STW1.Reserved13 := "DB_Drive_4UZ1".TelOut.STW1_BM.%X13;
   "HMI_DB".Drives.Drive_4UZ1.STW1.Reserved14 := "DB_Drive_4UZ1".TelOut.STW1_BM.%X14;
   "HMI_DB".Drives.Drive_4UZ1.STW1.Reserved15 := "DB_Drive_4UZ1".TelOut.STW1_BM.%X15;


   // ============================================================
   // 5. STW2_BM bits, PLC -> ПЧ
   // ============================================================

   "HMI_DB".Drives.Drive_4UZ1.STW2.Bit00 := "DB_Drive_4UZ1".TelOut.STW2_BM.%X0;
   "HMI_DB".Drives.Drive_4UZ1.STW2.Bit01 := "DB_Drive_4UZ1".TelOut.STW2_BM.%X1;
   "HMI_DB".Drives.Drive_4UZ1.STW2.Bit02 := "DB_Drive_4UZ1".TelOut.STW2_BM.%X2;
   "HMI_DB".Drives.Drive_4UZ1.STW2.Bit03 := "DB_Drive_4UZ1".TelOut.STW2_BM.%X3;
   "HMI_DB".Drives.Drive_4UZ1.STW2.Bit04 := "DB_Drive_4UZ1".TelOut.STW2_BM.%X4;
   "HMI_DB".Drives.Drive_4UZ1.STW2.Bit05 := "DB_Drive_4UZ1".TelOut.STW2_BM.%X5;
   "HMI_DB".Drives.Drive_4UZ1.STW2.Bit06 := "DB_Drive_4UZ1".TelOut.STW2_BM.%X6;
   "HMI_DB".Drives.Drive_4UZ1.STW2.Bit07 := "DB_Drive_4UZ1".TelOut.STW2_BM.%X7;
   "HMI_DB".Drives.Drive_4UZ1.STW2.Bit08 := "DB_Drive_4UZ1".TelOut.STW2_BM.%X8;
   "HMI_DB".Drives.Drive_4UZ1.STW2.Bit09 := "DB_Drive_4UZ1".TelOut.STW2_BM.%X9;
   "HMI_DB".Drives.Drive_4UZ1.STW2.Bit10 := "DB_Drive_4UZ1".TelOut.STW2_BM.%X10;
   "HMI_DB".Drives.Drive_4UZ1.STW2.Bit11 := "DB_Drive_4UZ1".TelOut.STW2_BM.%X11;
   "HMI_DB".Drives.Drive_4UZ1.STW2.Bit12 := "DB_Drive_4UZ1".TelOut.STW2_BM.%X12;
   "HMI_DB".Drives.Drive_4UZ1.STW2.Bit13 := "DB_Drive_4UZ1".TelOut.STW2_BM.%X13;
   "HMI_DB".Drives.Drive_4UZ1.STW2.Bit14 := "DB_Drive_4UZ1".TelOut.STW2_BM.%X14;
   "HMI_DB".Drives.Drive_4UZ1.STW2.Bit15 := "DB_Drive_4UZ1".TelOut.STW2_BM.%X15;


   // ============================================================
   // 6. ZSW1_BM bits, ПЧ -> PLC
   // ============================================================

   "HMI_DB".Drives.Drive_4UZ1.ZSW1.ReadyToSwitchOn := "DB_Drive_4UZ1".TelIn.ZSW1_BM.%X0;
   "HMI_DB".Drives.Drive_4UZ1.ZSW1.ReadyToOperate := "DB_Drive_4UZ1".TelIn.ZSW1_BM.%X1;
   "HMI_DB".Drives.Drive_4UZ1.ZSW1.OperationEnabled := "DB_Drive_4UZ1".TelIn.ZSW1_BM.%X2;
   "HMI_DB".Drives.Drive_4UZ1.ZSW1.FaultActive := "DB_Drive_4UZ1".TelIn.ZSW1_BM.%X3;
   "HMI_DB".Drives.Drive_4UZ1.ZSW1.NoCoastStopActive := "DB_Drive_4UZ1".TelIn.ZSW1_BM.%X4;
   "HMI_DB".Drives.Drive_4UZ1.ZSW1.NoQuickStopActive := "DB_Drive_4UZ1".TelIn.ZSW1_BM.%X5;
   "HMI_DB".Drives.Drive_4UZ1.ZSW1.SwitchingOnInhibit := "DB_Drive_4UZ1".TelIn.ZSW1_BM.%X6;
   "HMI_DB".Drives.Drive_4UZ1.ZSW1.WarningActive := "DB_Drive_4UZ1".TelIn.ZSW1_BM.%X7;
   "HMI_DB".Drives.Drive_4UZ1.ZSW1.SpeedErrorInTolerance := "DB_Drive_4UZ1".TelIn.ZSW1_BM.%X8;
   "HMI_DB".Drives.Drive_4UZ1.ZSW1.ControlRequested := "DB_Drive_4UZ1".TelIn.ZSW1_BM.%X9;
   "HMI_DB".Drives.Drive_4UZ1.ZSW1.SetpointReached := "DB_Drive_4UZ1".TelIn.ZSW1_BM.%X10;
   "HMI_DB".Drives.Drive_4UZ1.ZSW1.InternalLimitActive := "DB_Drive_4UZ1".TelIn.ZSW1_BM.%X11;
   "HMI_DB".Drives.Drive_4UZ1.ZSW1.Reserved12 := "DB_Drive_4UZ1".TelIn.ZSW1_BM.%X12;
   "HMI_DB".Drives.Drive_4UZ1.ZSW1.Reserved13 := "DB_Drive_4UZ1".TelIn.ZSW1_BM.%X13;
   "HMI_DB".Drives.Drive_4UZ1.ZSW1.Reserved14 := "DB_Drive_4UZ1".TelIn.ZSW1_BM.%X14;
   "HMI_DB".Drives.Drive_4UZ1.ZSW1.Reserved15 := "DB_Drive_4UZ1".TelIn.ZSW1_BM.%X15;


   // ============================================================
   // 7. ZSW2_BM bits, ПЧ -> PLC
   // ============================================================

   "HMI_DB".Drives.Drive_4UZ1.ZSW2.Bit00 := "DB_Drive_4UZ1".TelIn.ZSW2_BM.%X0;
   "HMI_DB".Drives.Drive_4UZ1.ZSW2.Bit01 := "DB_Drive_4UZ1".TelIn.ZSW2_BM.%X1;
   "HMI_DB".Drives.Drive_4UZ1.ZSW2.Bit02 := "DB_Drive_4UZ1".TelIn.ZSW2_BM.%X2;
   "HMI_DB".Drives.Drive_4UZ1.ZSW2.Bit03 := "DB_Drive_4UZ1".TelIn.ZSW2_BM.%X3;
   "HMI_DB".Drives.Drive_4UZ1.ZSW2.Bit04 := "DB_Drive_4UZ1".TelIn.ZSW2_BM.%X4;
   "HMI_DB".Drives.Drive_4UZ1.ZSW2.Bit05 := "DB_Drive_4UZ1".TelIn.ZSW2_BM.%X5;
   "HMI_DB".Drives.Drive_4UZ1.ZSW2.Bit06 := "DB_Drive_4UZ1".TelIn.ZSW2_BM.%X6;
   "HMI_DB".Drives.Drive_4UZ1.ZSW2.Bit07 := "DB_Drive_4UZ1".TelIn.ZSW2_BM.%X7;
   "HMI_DB".Drives.Drive_4UZ1.ZSW2.Bit08 := "DB_Drive_4UZ1".TelIn.ZSW2_BM.%X8;
   "HMI_DB".Drives.Drive_4UZ1.ZSW2.Bit09 := "DB_Drive_4UZ1".TelIn.ZSW2_BM.%X9;
   "HMI_DB".Drives.Drive_4UZ1.ZSW2.Bit10 := "DB_Drive_4UZ1".TelIn.ZSW2_BM.%X10;
   "HMI_DB".Drives.Drive_4UZ1.ZSW2.Bit11 := "DB_Drive_4UZ1".TelIn.ZSW2_BM.%X11;
   "HMI_DB".Drives.Drive_4UZ1.ZSW2.Bit12 := "DB_Drive_4UZ1".TelIn.ZSW2_BM.%X12;
   "HMI_DB".Drives.Drive_4UZ1.ZSW2.Bit13 := "DB_Drive_4UZ1".TelIn.ZSW2_BM.%X13;
   "HMI_DB".Drives.Drive_4UZ1.ZSW2.Bit14 := "DB_Drive_4UZ1".TelIn.ZSW2_BM.%X14;
   "HMI_DB".Drives.Drive_4UZ1.ZSW2.Bit15 := "DB_Drive_4UZ1".TelIn.ZSW2_BM.%X15;


   // ============================================================
   // 8. BRAKE_STATUS / r1229 bits, ПЧ -> PLC
   // ============================================================

   "HMI_DB".Drives.Drive_4UZ1.Brake.RawWord := "DB_Drive_4UZ1".TelIn.BRAKE_STATUS;

   "HMI_DB".Drives.Drive_4UZ1.Brake.Bit00 := "DB_Drive_4UZ1".TelIn.BRAKE_STATUS.%X0;
   "HMI_DB".Drives.Drive_4UZ1.Brake.CommandOpenBrake := "DB_Drive_4UZ1".TelIn.BRAKE_STATUS.%X1;
   "HMI_DB".Drives.Drive_4UZ1.Brake.Bit02 := "DB_Drive_4UZ1".TelIn.BRAKE_STATUS.%X2;
   "HMI_DB".Drives.Drive_4UZ1.Brake.PulseEnableExtendedBrakeControl := "DB_Drive_4UZ1".TelIn.BRAKE_STATUS.%X3;
   "HMI_DB".Drives.Drive_4UZ1.Brake.BrakeDoesNotOpen := "DB_Drive_4UZ1".TelIn.BRAKE_STATUS.%X4;
   "HMI_DB".Drives.Drive_4UZ1.Brake.BrakeDoesNotClose := "DB_Drive_4UZ1".TelIn.BRAKE_STATUS.%X5;
   "HMI_DB".Drives.Drive_4UZ1.Brake.BrakeThresholdExceeded := "DB_Drive_4UZ1".TelIn.BRAKE_STATUS.%X6;
   "HMI_DB".Drives.Drive_4UZ1.Brake.BrakeThresholdUndershot := "DB_Drive_4UZ1".TelIn.BRAKE_STATUS.%X7;
   "HMI_DB".Drives.Drive_4UZ1.Brake.BrakeMonitoringTimeExpired := "DB_Drive_4UZ1".TelIn.BRAKE_STATUS.%X8;
   "HMI_DB".Drives.Drive_4UZ1.Brake.PulseEnableRequestMissing := "DB_Drive_4UZ1".TelIn.BRAKE_STATUS.%X9;
   "HMI_DB".Drives.Drive_4UZ1.Brake.BrakeOrLogicResult := "DB_Drive_4UZ1".TelIn.BRAKE_STATUS.%X10;
   "HMI_DB".Drives.Drive_4UZ1.Brake.BrakeAndLogicResult := "DB_Drive_4UZ1".TelIn.BRAKE_STATUS.%X11;
   "HMI_DB".Drives.Drive_4UZ1.Brake.Bit12 := "DB_Drive_4UZ1".TelIn.BRAKE_STATUS.%X12;
   "HMI_DB".Drives.Drive_4UZ1.Brake.Bit13 := "DB_Drive_4UZ1".TelIn.BRAKE_STATUS.%X13;
   "HMI_DB".Drives.Drive_4UZ1.Brake.Bit14 := "DB_Drive_4UZ1".TelIn.BRAKE_STATUS.%X14;
   "HMI_DB".Drives.Drive_4UZ1.Brake.Bit15 := "DB_Drive_4UZ1".TelIn.BRAKE_STATUS.%X15;
END_REGION

REGION Network 5 (SCL): Копіювання даних ПЧ 4UZ2 на візуалізацію
   // ============================================================
   // 1. Основні значення та діагностика драйвера
   // ============================================================

   "HMI_DB".Drives.Drive_4UZ2.Values.AxisEnabled := "DB_Drive_4UZ2".AxisEnabled;
   "HMI_DB".Drives.Drive_4UZ2.Values.Lockout := "DB_Drive_4UZ2".Lockout;
   "HMI_DB".Drives.Drive_4UZ2.Values.Error := "DB_Drive_4UZ2".Error;
   "HMI_DB".Drives.Drive_4UZ2.Values.BrakeOpenRequest := "DB_Drive_4UZ2".BrakeOpenRequest;

   "HMI_DB".Drives.Drive_4UZ2.Values.ActVelocity_Rpm := "DB_Drive_4UZ2".ActVelocity;
   "HMI_DB".Drives.Drive_4UZ2.Values.SpeedSetpointFb_Rpm := "DB_Drive_4UZ2".SpeedSetpointFb;
   "HMI_DB".Drives.Drive_4UZ2.Values.ActCurrent_A := "DB_Drive_4UZ2".ActCurrent;
   "HMI_DB".Drives.Drive_4UZ2.Values.ActTorque_Nm := "DB_Drive_4UZ2".ActTorque;
   "HMI_DB".Drives.Drive_4UZ2.Values.ActPower_kW := "DB_Drive_4UZ2".ActPower;
   "HMI_DB".Drives.Drive_4UZ2.Values.LoadPower_Pct := "DB_Drive_4UZ2".LoadPower;

   "HMI_DB".Drives.Drive_4UZ2.Values.FaultCode := "DB_Drive_4UZ2".FaultCode;
   "HMI_DB".Drives.Drive_4UZ2.Values.WarningCode := "DB_Drive_4UZ2".WarningCode;
   "HMI_DB".Drives.Drive_4UZ2.Values.Status := "DB_Drive_4UZ2".Status;
   "HMI_DB".Drives.Drive_4UZ2.Values.DiagId := "DB_Drive_4UZ2".DiagId;

   "HMI_DB".Drives.Drive_4UZ2.Values.SpeedError_Rpm := "DB_Drive_4UZ2".SpeedSetpointFb - "DB_Drive_4UZ2".ActVelocity;

   // ============================================================
   // Status driver bits
   // ============================================================

   "HMI_DB".Drives.Drive_4UZ2.StatusBits.ReadOk := "DB_Drive_4UZ2".Status.%X0;
   "HMI_DB".Drives.Drive_4UZ2.StatusBits.WriteOk := "DB_Drive_4UZ2".Status.%X1;
   "HMI_DB".Drives.Drive_4UZ2.StatusBits.AxisEnabled := "DB_Drive_4UZ2".Status.%X2;
   "HMI_DB".Drives.Drive_4UZ2.StatusBits.Lockout := "DB_Drive_4UZ2".Status.%X3;
   "HMI_DB".Drives.Drive_4UZ2.StatusBits.DriveFault := "DB_Drive_4UZ2".Status.%X4;
   "HMI_DB".Drives.Drive_4UZ2.StatusBits.DriveWarning := "DB_Drive_4UZ2".Status.%X5;
   "HMI_DB".Drives.Drive_4UZ2.StatusBits.BrakeOpenRequest := "DB_Drive_4UZ2".Status.%X6;
   "HMI_DB".Drives.Drive_4UZ2.StatusBits.SimMode := "DB_Drive_4UZ2".Status.%X7;
   "HMI_DB".Drives.Drive_4UZ2.StatusBits.SwitchingOnInhibit := "DB_Drive_4UZ2".Status.%X8;
   "HMI_DB".Drives.Drive_4UZ2.StatusBits.ControlRequested := "DB_Drive_4UZ2".Status.%X9;
   "HMI_DB".Drives.Drive_4UZ2.StatusBits.Reserved10 := "DB_Drive_4UZ2".Status.%X10;
   "HMI_DB".Drives.Drive_4UZ2.StatusBits.Reserved11 := "DB_Drive_4UZ2".Status.%X11;
   "HMI_DB".Drives.Drive_4UZ2.StatusBits.Reserved12 := "DB_Drive_4UZ2".Status.%X12;
   "HMI_DB".Drives.Drive_4UZ2.StatusBits.Reserved13 := "DB_Drive_4UZ2".Status.%X13;
   "HMI_DB".Drives.Drive_4UZ2.StatusBits.Reserved14 := "DB_Drive_4UZ2".Status.%X14;
   "HMI_DB".Drives.Drive_4UZ2.StatusBits.Reserved15 := "DB_Drive_4UZ2".Status.%X15;

   // ============================================================
   // 2. Raw telegram PLC -> ПЧ
   // ============================================================

   "HMI_DB".Drives.Drive_4UZ2.Raw.STW1_BM := "DB_Drive_4UZ2".TelOut.STW1_BM;
   "HMI_DB".Drives.Drive_4UZ2.Raw.NSOLL_B := "DB_Drive_4UZ2".TelOut.NSOLL_B;
   "HMI_DB".Drives.Drive_4UZ2.Raw.STW2_BM := "DB_Drive_4UZ2".TelOut.STW2_BM;
   "HMI_DB".Drives.Drive_4UZ2.Raw.M_ADD := "DB_Drive_4UZ2".TelOut.M_ADD;
   "HMI_DB".Drives.Drive_4UZ2.Raw.M_LIM := "DB_Drive_4UZ2".TelOut.M_LIM;
   "HMI_DB".Drives.Drive_4UZ2.Raw.USER_1 := "DB_Drive_4UZ2".TelOut.USER_1;
   "HMI_DB".Drives.Drive_4UZ2.Raw.USER_2 := "DB_Drive_4UZ2".TelOut.USER_2;
   "HMI_DB".Drives.Drive_4UZ2.Raw.USER_3 := "DB_Drive_4UZ2".TelOut.USER_3;
   "HMI_DB".Drives.Drive_4UZ2.Raw.USER_4 := "DB_Drive_4UZ2".TelOut.USER_4;



   // ============================================================
   // 3. Raw telegram ПЧ -> PLC
   // ============================================================

   "HMI_DB".Drives.Drive_4UZ2.Raw.ZSW1_BM := "DB_Drive_4UZ2".TelIn.ZSW1_BM;
   "HMI_DB".Drives.Drive_4UZ2.Raw.NIST_A := "DB_Drive_4UZ2".TelIn.NIST_A;
   "HMI_DB".Drives.Drive_4UZ2.Raw.IAIST := "DB_Drive_4UZ2".TelIn.IAIST;
   "HMI_DB".Drives.Drive_4UZ2.Raw.MIST := "DB_Drive_4UZ2".TelIn.MIST;
   "HMI_DB".Drives.Drive_4UZ2.Raw.WARN_CODE := "DB_Drive_4UZ2".TelIn.WARN_CODE;
   "HMI_DB".Drives.Drive_4UZ2.Raw.FAULT_CODE := "DB_Drive_4UZ2".TelIn.FAULT_CODE;
   "HMI_DB".Drives.Drive_4UZ2.Raw.ZSW2_BM := "DB_Drive_4UZ2".TelIn.ZSW2_BM;
   "HMI_DB".Drives.Drive_4UZ2.Raw.NSET_FB := "DB_Drive_4UZ2".TelIn.NSET_FB;
   "HMI_DB".Drives.Drive_4UZ2.Raw.P_ACT := "DB_Drive_4UZ2".TelIn.P_ACT;
   "HMI_DB".Drives.Drive_4UZ2.Raw.BRAKE_STATUS := "DB_Drive_4UZ2".TelIn.BRAKE_STATUS;


   // ============================================================
   // 4. STW1_BM bits, PLC -> ПЧ
   // ============================================================

   "HMI_DB".Drives.Drive_4UZ2.STW1.OnOff1 := "DB_Drive_4UZ2".TelOut.STW1_BM.%X0;
   "HMI_DB".Drives.Drive_4UZ2.STW1.NoCoastStop := "DB_Drive_4UZ2".TelOut.STW1_BM.%X1;
   "HMI_DB".Drives.Drive_4UZ2.STW1.NoQuickStop := "DB_Drive_4UZ2".TelOut.STW1_BM.%X2;
   "HMI_DB".Drives.Drive_4UZ2.STW1.EnableOperation := "DB_Drive_4UZ2".TelOut.STW1_BM.%X3;
   "HMI_DB".Drives.Drive_4UZ2.STW1.RampGeneratorEnable := "DB_Drive_4UZ2".TelOut.STW1_BM.%X4;
   "HMI_DB".Drives.Drive_4UZ2.STW1.RampGeneratorContinue := "DB_Drive_4UZ2".TelOut.STW1_BM.%X5;
   "HMI_DB".Drives.Drive_4UZ2.STW1.SetpointEnable := "DB_Drive_4UZ2".TelOut.STW1_BM.%X6;
   "HMI_DB".Drives.Drive_4UZ2.STW1.FaultAcknowledge := "DB_Drive_4UZ2".TelOut.STW1_BM.%X7;
   "HMI_DB".Drives.Drive_4UZ2.STW1.Reserved08 := "DB_Drive_4UZ2".TelOut.STW1_BM.%X8;
   "HMI_DB".Drives.Drive_4UZ2.STW1.Reserved09 := "DB_Drive_4UZ2".TelOut.STW1_BM.%X9;
   "HMI_DB".Drives.Drive_4UZ2.STW1.ControlByPLC := "DB_Drive_4UZ2".TelOut.STW1_BM.%X10;
   "HMI_DB".Drives.Drive_4UZ2.STW1.Reserved11 := "DB_Drive_4UZ2".TelOut.STW1_BM.%X11;
   "HMI_DB".Drives.Drive_4UZ2.STW1.Reserved12 := "DB_Drive_4UZ2".TelOut.STW1_BM.%X12;
   "HMI_DB".Drives.Drive_4UZ2.STW1.Reserved13 := "DB_Drive_4UZ2".TelOut.STW1_BM.%X13;
   "HMI_DB".Drives.Drive_4UZ2.STW1.Reserved14 := "DB_Drive_4UZ2".TelOut.STW1_BM.%X14;
   "HMI_DB".Drives.Drive_4UZ2.STW1.Reserved15 := "DB_Drive_4UZ2".TelOut.STW1_BM.%X15;


   // ============================================================
   // 5. STW2_BM bits, PLC -> ПЧ
   // ============================================================

   "HMI_DB".Drives.Drive_4UZ2.STW2.Bit00 := "DB_Drive_4UZ2".TelOut.STW2_BM.%X0;
   "HMI_DB".Drives.Drive_4UZ2.STW2.Bit01 := "DB_Drive_4UZ2".TelOut.STW2_BM.%X1;
   "HMI_DB".Drives.Drive_4UZ2.STW2.Bit02 := "DB_Drive_4UZ2".TelOut.STW2_BM.%X2;
   "HMI_DB".Drives.Drive_4UZ2.STW2.Bit03 := "DB_Drive_4UZ2".TelOut.STW2_BM.%X3;
   "HMI_DB".Drives.Drive_4UZ2.STW2.Bit04 := "DB_Drive_4UZ2".TelOut.STW2_BM.%X4;
   "HMI_DB".Drives.Drive_4UZ2.STW2.Bit05 := "DB_Drive_4UZ2".TelOut.STW2_BM.%X5;
   "HMI_DB".Drives.Drive_4UZ2.STW2.Bit06 := "DB_Drive_4UZ2".TelOut.STW2_BM.%X6;
   "HMI_DB".Drives.Drive_4UZ2.STW2.Bit07 := "DB_Drive_4UZ2".TelOut.STW2_BM.%X7;
   "HMI_DB".Drives.Drive_4UZ2.STW2.Bit08 := "DB_Drive_4UZ2".TelOut.STW2_BM.%X8;
   "HMI_DB".Drives.Drive_4UZ2.STW2.Bit09 := "DB_Drive_4UZ2".TelOut.STW2_BM.%X9;
   "HMI_DB".Drives.Drive_4UZ2.STW2.Bit10 := "DB_Drive_4UZ2".TelOut.STW2_BM.%X10;
   "HMI_DB".Drives.Drive_4UZ2.STW2.Bit11 := "DB_Drive_4UZ2".TelOut.STW2_BM.%X11;
   "HMI_DB".Drives.Drive_4UZ2.STW2.Bit12 := "DB_Drive_4UZ2".TelOut.STW2_BM.%X12;
   "HMI_DB".Drives.Drive_4UZ2.STW2.Bit13 := "DB_Drive_4UZ2".TelOut.STW2_BM.%X13;
   "HMI_DB".Drives.Drive_4UZ2.STW2.Bit14 := "DB_Drive_4UZ2".TelOut.STW2_BM.%X14;
   "HMI_DB".Drives.Drive_4UZ2.STW2.Bit15 := "DB_Drive_4UZ2".TelOut.STW2_BM.%X15;


   // ============================================================
   // 6. ZSW1_BM bits, ПЧ -> PLC
   // ============================================================

   "HMI_DB".Drives.Drive_4UZ2.ZSW1.ReadyToSwitchOn := "DB_Drive_4UZ2".TelIn.ZSW1_BM.%X0;
   "HMI_DB".Drives.Drive_4UZ2.ZSW1.ReadyToOperate := "DB_Drive_4UZ2".TelIn.ZSW1_BM.%X1;
   "HMI_DB".Drives.Drive_4UZ2.ZSW1.OperationEnabled := "DB_Drive_4UZ2".TelIn.ZSW1_BM.%X2;
   "HMI_DB".Drives.Drive_4UZ2.ZSW1.FaultActive := "DB_Drive_4UZ2".TelIn.ZSW1_BM.%X3;
   "HMI_DB".Drives.Drive_4UZ2.ZSW1.NoCoastStopActive := "DB_Drive_4UZ2".TelIn.ZSW1_BM.%X4;
   "HMI_DB".Drives.Drive_4UZ2.ZSW1.NoQuickStopActive := "DB_Drive_4UZ2".TelIn.ZSW1_BM.%X5;
   "HMI_DB".Drives.Drive_4UZ2.ZSW1.SwitchingOnInhibit := "DB_Drive_4UZ2".TelIn.ZSW1_BM.%X6;
   "HMI_DB".Drives.Drive_4UZ2.ZSW1.WarningActive := "DB_Drive_4UZ2".TelIn.ZSW1_BM.%X7;
   "HMI_DB".Drives.Drive_4UZ2.ZSW1.SpeedErrorInTolerance := "DB_Drive_4UZ2".TelIn.ZSW1_BM.%X8;
   "HMI_DB".Drives.Drive_4UZ2.ZSW1.ControlRequested := "DB_Drive_4UZ2".TelIn.ZSW1_BM.%X9;
   "HMI_DB".Drives.Drive_4UZ2.ZSW1.SetpointReached := "DB_Drive_4UZ2".TelIn.ZSW1_BM.%X10;
   "HMI_DB".Drives.Drive_4UZ2.ZSW1.InternalLimitActive := "DB_Drive_4UZ2".TelIn.ZSW1_BM.%X11;
   "HMI_DB".Drives.Drive_4UZ2.ZSW1.Reserved12 := "DB_Drive_4UZ2".TelIn.ZSW1_BM.%X12;
   "HMI_DB".Drives.Drive_4UZ2.ZSW1.Reserved13 := "DB_Drive_4UZ2".TelIn.ZSW1_BM.%X13;
   "HMI_DB".Drives.Drive_4UZ2.ZSW1.Reserved14 := "DB_Drive_4UZ2".TelIn.ZSW1_BM.%X14;
   "HMI_DB".Drives.Drive_4UZ2.ZSW1.Reserved15 := "DB_Drive_4UZ2".TelIn.ZSW1_BM.%X15;


   // ============================================================
   // 7. ZSW2_BM bits, ПЧ -> PLC
   // ============================================================

   "HMI_DB".Drives.Drive_4UZ2.ZSW2.Bit00 := "DB_Drive_4UZ2".TelIn.ZSW2_BM.%X0;
   "HMI_DB".Drives.Drive_4UZ2.ZSW2.Bit01 := "DB_Drive_4UZ2".TelIn.ZSW2_BM.%X1;
   "HMI_DB".Drives.Drive_4UZ2.ZSW2.Bit02 := "DB_Drive_4UZ2".TelIn.ZSW2_BM.%X2;
   "HMI_DB".Drives.Drive_4UZ2.ZSW2.Bit03 := "DB_Drive_4UZ2".TelIn.ZSW2_BM.%X3;
   "HMI_DB".Drives.Drive_4UZ2.ZSW2.Bit04 := "DB_Drive_4UZ2".TelIn.ZSW2_BM.%X4;
   "HMI_DB".Drives.Drive_4UZ2.ZSW2.Bit05 := "DB_Drive_4UZ2".TelIn.ZSW2_BM.%X5;
   "HMI_DB".Drives.Drive_4UZ2.ZSW2.Bit06 := "DB_Drive_4UZ2".TelIn.ZSW2_BM.%X6;
   "HMI_DB".Drives.Drive_4UZ2.ZSW2.Bit07 := "DB_Drive_4UZ2".TelIn.ZSW2_BM.%X7;
   "HMI_DB".Drives.Drive_4UZ2.ZSW2.Bit08 := "DB_Drive_4UZ2".TelIn.ZSW2_BM.%X8;
   "HMI_DB".Drives.Drive_4UZ2.ZSW2.Bit09 := "DB_Drive_4UZ2".TelIn.ZSW2_BM.%X9;
   "HMI_DB".Drives.Drive_4UZ2.ZSW2.Bit10 := "DB_Drive_4UZ2".TelIn.ZSW2_BM.%X10;
   "HMI_DB".Drives.Drive_4UZ2.ZSW2.Bit11 := "DB_Drive_4UZ2".TelIn.ZSW2_BM.%X11;
   "HMI_DB".Drives.Drive_4UZ2.ZSW2.Bit12 := "DB_Drive_4UZ2".TelIn.ZSW2_BM.%X12;
   "HMI_DB".Drives.Drive_4UZ2.ZSW2.Bit13 := "DB_Drive_4UZ2".TelIn.ZSW2_BM.%X13;
   "HMI_DB".Drives.Drive_4UZ2.ZSW2.Bit14 := "DB_Drive_4UZ2".TelIn.ZSW2_BM.%X14;
   "HMI_DB".Drives.Drive_4UZ2.ZSW2.Bit15 := "DB_Drive_4UZ2".TelIn.ZSW2_BM.%X15;


   // ============================================================
   // 8. BRAKE_STATUS / r1229 bits, ПЧ -> PLC
   // ============================================================

   "HMI_DB".Drives.Drive_4UZ2.Brake.RawWord := "DB_Drive_4UZ2".TelIn.BRAKE_STATUS;

   "HMI_DB".Drives.Drive_4UZ2.Brake.Bit00 := "DB_Drive_4UZ2".TelIn.BRAKE_STATUS.%X0;
   "HMI_DB".Drives.Drive_4UZ2.Brake.CommandOpenBrake := "DB_Drive_4UZ2".TelIn.BRAKE_STATUS.%X1;
   "HMI_DB".Drives.Drive_4UZ2.Brake.Bit02 := "DB_Drive_4UZ2".TelIn.BRAKE_STATUS.%X2;
   "HMI_DB".Drives.Drive_4UZ2.Brake.PulseEnableExtendedBrakeControl := "DB_Drive_4UZ2".TelIn.BRAKE_STATUS.%X3;
   "HMI_DB".Drives.Drive_4UZ2.Brake.BrakeDoesNotOpen := "DB_Drive_4UZ2".TelIn.BRAKE_STATUS.%X4;
   "HMI_DB".Drives.Drive_4UZ2.Brake.BrakeDoesNotClose := "DB_Drive_4UZ2".TelIn.BRAKE_STATUS.%X5;
   "HMI_DB".Drives.Drive_4UZ2.Brake.BrakeThresholdExceeded := "DB_Drive_4UZ2".TelIn.BRAKE_STATUS.%X6;
   "HMI_DB".Drives.Drive_4UZ2.Brake.BrakeThresholdUndershot := "DB_Drive_4UZ2".TelIn.BRAKE_STATUS.%X7;
   "HMI_DB".Drives.Drive_4UZ2.Brake.BrakeMonitoringTimeExpired := "DB_Drive_4UZ2".TelIn.BRAKE_STATUS.%X8;
   "HMI_DB".Drives.Drive_4UZ2.Brake.PulseEnableRequestMissing := "DB_Drive_4UZ2".TelIn.BRAKE_STATUS.%X9;
   "HMI_DB".Drives.Drive_4UZ2.Brake.BrakeOrLogicResult := "DB_Drive_4UZ2".TelIn.BRAKE_STATUS.%X10;
   "HMI_DB".Drives.Drive_4UZ2.Brake.BrakeAndLogicResult := "DB_Drive_4UZ2".TelIn.BRAKE_STATUS.%X11;
   "HMI_DB".Drives.Drive_4UZ2.Brake.Bit12 := "DB_Drive_4UZ2".TelIn.BRAKE_STATUS.%X12;
   "HMI_DB".Drives.Drive_4UZ2.Brake.Bit13 := "DB_Drive_4UZ2".TelIn.BRAKE_STATUS.%X13;
   "HMI_DB".Drives.Drive_4UZ2.Brake.Bit14 := "DB_Drive_4UZ2".TelIn.BRAKE_STATUS.%X14;
   "HMI_DB".Drives.Drive_4UZ2.Brake.Bit15 := "DB_Drive_4UZ2".TelIn.BRAKE_STATUS.%X15;
END_REGION
END_FUNCTION

FUNCTION "FC_CU_U1_HMI" : Void   // FC52, LAD
{ S7_Optimized_Access := 'TRUE' }
VERSION : 0.1
BEGIN

REGION Network 2 (SCL): Дані на HMI для блока управління приводами U1 CU320-2 PN
   // ============================================================
   // 1. Основні значення та діагностика CU
   // ============================================================

   "HMI_DB".Drives.CU_U1.Values.CommOk := "DB_CU_U1".CommOk;
   "HMI_DB".Drives.CU_U1.Values.Fault := "DB_CU_U1".Fault;
   "HMI_DB".Drives.CU_U1.Values.Warning := "DB_CU_U1".Warning;
   "HMI_DB".Drives.CU_U1.Values.Error := "DB_CU_U1".Error;

   "HMI_DB".Drives.CU_U1.Values.CU_StatusWord := "DB_CU_U1".CU_StatusWord;
   "HMI_DB".Drives.CU_U1.Values.CU_DiagCode := "DB_CU_U1".CU_DiagCode;

   "HMI_DB".Drives.CU_U1.Values.Status := "DB_CU_U1".Status;
   "HMI_DB".Drives.CU_U1.Values.DiagId := "DB_CU_U1".DiagId;


   // ============================================================
   // 2. Status driver bits
   // ============================================================

   "HMI_DB".Drives.CU_U1.StatusBits.ReadOk := "DB_CU_U1".Status.%X0;
   "HMI_DB".Drives.CU_U1.StatusBits.WriteOk := "DB_CU_U1".Status.%X1;
   "HMI_DB".Drives.CU_U1.StatusBits.CommOk := "DB_CU_U1".Status.%X2;
   "HMI_DB".Drives.CU_U1.StatusBits.Fault := "DB_CU_U1".Status.%X3;
   "HMI_DB".Drives.CU_U1.StatusBits.Warning := "DB_CU_U1".Status.%X4;
   "HMI_DB".Drives.CU_U1.StatusBits.SwitchingOnInhibit := "DB_CU_U1".Status.%X5;
   "HMI_DB".Drives.CU_U1.StatusBits.ControlRequested := "DB_CU_U1".Status.%X6;
   "HMI_DB".Drives.CU_U1.StatusBits.SimMode := "DB_CU_U1".Status.%X7;
   "HMI_DB".Drives.CU_U1.StatusBits.Reserved08 := "DB_CU_U1".Status.%X8;
   "HMI_DB".Drives.CU_U1.StatusBits.Reserved09 := "DB_CU_U1".Status.%X9;
   "HMI_DB".Drives.CU_U1.StatusBits.Reserved10 := "DB_CU_U1".Status.%X10;
   "HMI_DB".Drives.CU_U1.StatusBits.Reserved11 := "DB_CU_U1".Status.%X11;
   "HMI_DB".Drives.CU_U1.StatusBits.Reserved12 := "DB_CU_U1".Status.%X12;
   "HMI_DB".Drives.CU_U1.StatusBits.Reserved13 := "DB_CU_U1".Status.%X13;
   "HMI_DB".Drives.CU_U1.StatusBits.Reserved14 := "DB_CU_U1".Status.%X14;
   "HMI_DB".Drives.CU_U1.StatusBits.Reserved15 := "DB_CU_U1".Status.%X15;


   // ============================================================
   // 3. Raw telegram PLC -> CU
   // ============================================================

   "HMI_DB".Drives.CU_U1.Raw.CU_STW1 := "DB_CU_U1".TelOut.CU_STW1;
   "HMI_DB".Drives.CU_U1.Raw.CU_CTRL2 := "DB_CU_U1".TelOut.CU_CTRL2;


   // ============================================================
   // 4. Raw telegram CU -> PLC
   // ============================================================

   "HMI_DB".Drives.CU_U1.Raw.CU_ZSW1 := "DB_CU_U1".TelIn.CU_ZSW1;
   "HMI_DB".Drives.CU_U1.Raw.CU_DIAG_CODE := "DB_CU_U1".TelIn.CU_DIAG_CODE;


   // ============================================================
   // 5. CU_STW1 bits, PLC -> CU
   // ============================================================

